LIN {X 0,Y 362.16,Z 503.994,A -85,B 0,C 180,E1 -13146.687,E2 -13146.687} C_VEL
LIN {X 0,Y 362.023,Z 504.013,A -85,B 0,C 180,E1 -13150.063,E2 -13150.063} C_VEL
LIN {X 0,Y 361.989,Z 504.018,A -85,B 0,C 180,E1 -13153.9,E2 -13153.9} C_VEL
LIN {X 0,Y 361.959,Z 504.022,A -85,B 0,C 180,E1 -13157.939,E2 -13157.939} C_VEL
LIN {X 0,Y 361.884,Z 504.034,A -85,B 0,C 180,E1 -13161.654,E2 -13161.654} C_VEL
LIN {X 0,Y 361.921,Z 504.028,A -85,B 0,C 180,E1 -13165.291,E2 -13165.291} C_VEL
LIN {X 0,Y 361.916,Z 504.029,A -85,B 0,C 180,E1 -13167.779,E2 -13167.779} C_VEL
LIN {X 0,Y 361.854,Z 504.038,A -85,B 0,C 180,E1 -13171.628,E2 -13171.628} C_VEL
LIN {X 0,Y 361.87,Z 504.035,A -85,B 0,C 180,E1 -13175.346,E2 -13175.346} C_VEL
LIN {X 0,Y 361.871,Z 504.032,A -85,B 0,C 180,E1 -13179.029,E2 -13179.029} C_VEL
LIN {X 0,Y 361.883,Z 504.029,A -85,B 0,C 180,E1 -13182.442,E2 -13182.442} C_VEL
LIN {X 0,Y 361.926,Z 504.026,A -85,B 0,C 180,E1 -13185.93,E2 -13185.93} C_VEL
LIN {X 0,Y 361.904,Z 504.029,A -85,B 0,C 180,E1 -13189.233,E2 -13189.233} C_VEL
LIN {X 0,Y 361.869,Z 504.032,A -85,B 0,C 180,E1 -13192.984,E2 -13192.984} C_VEL
LIN {X 0,Y 361.858,Z 504.032,A -85,B 0,C 180,E1 -13196.632,E2 -13196.632} C_VEL
LIN {X 0,Y 361.875,Z 504.036,A -85,B 0,C 180,E1 -13199.673,E2 -13199.673} C_VEL
LIN {X 0,Y 361.956,Z 504.025,A -85,B 0,C 180,E1 -13203.476,E2 -13203.476} C_VEL
LIN {X 0,Y 361.893,Z 504.03,A -85,B 0,C 180,E1 -13207.146,E2 -13207.146} C_VEL
LIN {X 0,Y 361.924,Z 504.024,A -85,B 0,C 180,E1 -13210.725,E2 -13210.725} C_VEL
LIN {X 0,Y 361.95,Z 504.021,A -85,B 0,C 180,E1 -13214.227,E2 -13214.227} C_VEL
LIN {X 0,Y 362.002,Z 504.014,A -85,B 0,C 180,E1 -13216.529,E2 -13216.529} C_VEL
LIN {X 0,Y 362.032,Z 504.013,A -85,B 0,C 180,E1 -13219.939,E2 -13219.939} C_VEL
LIN {X 0,Y 362.156,Z 503.998,A -85,B 0,C 180,E1 -13223.314,E2 -13223.314} C_VEL
LIN {X 0,Y 362.288,Z 503.983,A -85,B 0,C 180,E1 -13227.777,E2 -13227.777} C_VEL
LIN {X 0,Y 362.429,Z 503.963,A -85,B 0,C 180,E1 -13230.001,E2 -13230.001} C_VEL
LIN {X 0,Y 362.09,Z 504.004,A -85,B 0,C 180,E1 -13232.225,E2 -13232.225} C_VEL
LIN {X 0,Y 361.698,Z 504.058,A -85,B 0,C 180,E1 -13235.576,E2 -13235.576} C_VEL
LIN {X 0,Y 361.473,Z 504.131,A -85,B 0,C 180,E1 -13237.437,E2 -13237.437} C_VEL
LIN {X 0,Y 361.189,Z 507.102,A -85,B 0,C 180,E1 -13241.221,E2 -13241.221} C_VEL
LIN {X 0,Y 361.205,Z 507.651,A -85,B 0,C 180,E1 -13241.824,E2 -13241.824} C_VEL
LIN {X 0,Y 362.214,Z 510.606,A -85,B 0,C 180,E1 -13241.986,E2 -13241.986} C_VEL
LIN {X 0,Y 367.763,Z 525.518,A -85,B 0,C 180,E1 -13242.934,E2 -13242.934} C_VEL
LIN {X 0,Y 372.106,Z 539.202,A -85,B 0,C 180,E1 -13243.935,E2 -13243.935} C_VEL
LIN {X 0,Y 374.364,Z 547.439,A -85,B 0,C 180,E1 -13244.603,E2 -13244.603} C_VEL
LIN {X 0,Y 373.094,Z 561.384,A -85,B 0,C 180,E1 -13245.548,E2 -13245.548} C_VEL
LIN {X 0,Y 371.697,Z 574.147,A -85,B 0,C 180,E1 -13246.618,E2 -13246.618} C_VEL
LIN {X 0,Y 370.152,Z 586.321,A -85,B 0,C 180,E1 -13247.851,E2 -13247.851} C_VEL
LIN {X 0,Y 368.527,Z 598.526,A -85,B 0,C 180,E1 -13249.351,E2 -13249.351} C_VEL
LIN {X 0,Y 366.709,Z 610.314,A -85,B 0,C 180,E1 -13251.093,E2 -13251.093} C_VEL
LIN {X 0,Y 365.196,Z 620.6,A -85,B 0,C 180,E1 -13252.936,E2 -13252.936} C_VEL
LIN {X 0,Y 363.887,Z 629.278,A -85,B 0,C 180,E1 -13254.803,E2 -13254.803} C_VEL
LIN {X 0,Y 362.73,Z 637.566,A -85,B 0,C 180,E1 -13256.966,E2 -13256.966} C_VEL
LIN {X 0,Y 361.854,Z 644.084,A -85,B 0,C 180,E1 -13259.072,E2 -13259.072} C_VEL
LIN {X 0,Y 361.248,Z 649.166,A -85,B 0,C 180,E1 -13261.127,E2 -13261.127} C_VEL
LIN {X 0,Y 360.827,Z 653.239,A -85,B 0,C 180,E1 -13263.257,E2 -13263.257} C_VEL
LIN {X 0,Y 359.954,Z 654.717,A -85,B 0,C 180,E1 -13264.16,E2 -13264.16} C_VEL
LIN {X 0,Y 356.859,Z 656.726,A -85,B 0,C 180,E1 -13265.63,E2 -13265.63} C_VEL
LIN {X 0,Y 354.342,Z 657.99,A -85,B 0,C 180,E1 -13266.829,E2 -13266.829} C_VEL
LIN {X 0,Y 353.271,Z 658.718,A -85,B 0,C 180,E1 -13267.765,E2 -13267.765} C_VEL
LIN {X 0,Y 353.185,Z 658.865,A -85,B 0,C 180,E1 -13268.083,E2 -13268.083} C_VEL
LIN {X 0,Y 353.136,Z 659.368,A -85,B 0,C 180,E1 -13269.558,E2 -13269.558} C_VEL
LIN {X 0,Y 353.143,Z 659.407,A -85,B 0,C 180,E1 -13271.052,E2 -13271.052} C_VEL
LIN {X 0,Y 353.242,Z 658.953,A -85,B 0,C 180,E1 -13272.595,E2 -13272.595} C_VEL
LIN {X 0,Y 353.396,Z 657.843,A -85,B 0,C 180,E1 -13274.279,E2 -13274.279} C_VEL
LIN {X 0,Y 353.643,Z 656.133,A -85,B 0,C 180,E1 -13275.927,E2 -13275.927} C_VEL
LIN {X 0,Y 354.153,Z 652.64,A -85,B 0,C 180,E1 -13278.28,E2 -13278.28} C_VEL
LIN {X 0,Y 354.854,Z 647.717,A -85,B 0,C 180,E1 -13280.67,E2 -13280.67} C_VEL
LIN {X 0,Y 355.849,Z 641.498,A -85,B 0,C 180,E1 -13282.987,E2 -13282.987} C_VEL
LIN {X 0,Y 357.13,Z 634.019,A -85,B 0,C 180,E1 -13285.201,E2 -13285.201} C_VEL
LIN {X 0,Y 358.47,Z 626.29,A -85,B 0,C 180,E1 -13287.087,E2 -13287.087} C_VEL
LIN {X 0,Y 360.334,Z 616.189,A -85,B 0,C 180,E1 -13289.112,E2 -13289.112} C_VEL
LIN {X 0,Y 362.146,Z 605.801,A -85,B 0,C 180,E1 -13290.843,E2 -13290.843} C_VEL
LIN {X 0,Y 364.021,Z 594.626,A -85,B 0,C 180,E1 -13292.395,E2 -13292.395} C_VEL
LIN {X 0,Y 365.803,Z 582.756,A -85,B 0,C 180,E1 -13293.775,E2 -13293.775} C_VEL
LIN {X 0,Y 367.569,Z 569.94,A -85,B 0,C 180,E1 -13295.002,E2 -13295.002} C_VEL
LIN {X 0,Y 369.207,Z 556.741,A -85,B 0,C 180,E1 -13296.021,E2 -13296.021} C_VEL
LIN {X 0,Y 369.669,Z 552.277,A -85,B 0,C 180,E1 -13296.32,E2 -13296.32} C_VEL
LIN {X 0,Y 368.858,Z 548.08,A -85,B 0,C 180,E1 -13296.697,E2 -13296.697} C_VEL
LIN {X 0,Y 364.908,Z 535.544,A -85,B 0,C 180,E1 -13297.833,E2 -13297.833} C_VEL
LIN {X 0,Y 359.987,Z 523.202,A -85,B 0,C 180,E1 -13298.919,E2 -13298.919} C_VEL
LIN {X 0,Y 355.705,Z 514.122,A -85,B 0,C 180,E1 -13299.696,E2 -13299.696} C_VEL
LIN {X 0,Y 354.522,Z 510.981,A -85,B 0,C 180,E1 -13299.927,E2 -13299.927} C_VEL
LIN {X 0,Y 354.688,Z 509.194,A -85,B 0,C 180,E1 -13302.709,E2 -13302.709} C_VEL
LIN {X 0,Y 354.966,Z 507.016,A -85,B 0,C 180,E1 -13306.255,E2 -13306.255} C_VEL
LIN {X 0,Y 354.941,Z 505.058,A -85,B 0,C 180,E1 -13309.734,E2 -13309.734} C_VEL
LIN {X 0,Y 355.125,Z 504.875,A -85,B 0,C 180,E1 -13313.18,E2 -13313.18} C_VEL
LIN {X 0,Y 355.244,Z 504.861,A -85,B 0,C 180,E1 -13317.732,E2 -13317.732} C_VEL
LIN {X 0,Y 355.395,Z 504.84,A -85,B 0,C 180,E1 -13320,E2 -13320} C_VEL
LIN {X 0,Y 355.243,Z 504.86,A -85,B 0,C 180,E1 -13322.267,E2 -13322.267} C_VEL
LIN {X 0,Y 355.136,Z 504.873,A -85,B 0,C 180,E1 -13326.819,E2 -13326.819} C_VEL
LIN {X 0,Y 355.013,Z 504.887,A -85,B 0,C 180,E1 -13329.112,E2 -13329.112} C_VEL
LIN {X 0,Y 354.918,Z 504.902,A -85,B 0,C 180,E1 -13332.581,E2 -13332.581} C_VEL
LIN {X 0,Y 354.886,Z 504.903,A -85,B 0,C 180,E1 -13336.096,E2 -13336.096} C_VEL
LIN {X 0,Y 354.9,Z 504.905,A -85,B 0,C 180,E1 -13338.472,E2 -13338.472} C_VEL
LIN {X 0,Y 354.832,Z 504.911,A -85,B 0,C 180,E1 -13342.106,E2 -13342.106} C_VEL
LIN {X 0,Y 354.897,Z 504.904,A -85,B 0,C 180,E1 -13345.827,E2 -13345.827} C_VEL
LIN {X 0,Y 354.852,Z 504.91,A -85,B 0,C 180,E1 -13349.678,E2 -13349.678} C_VEL
LIN {X 0,Y 354.784,Z 504.919,A -85,B 0,C 180,E1 -13352.333,E2 -13352.333} C_VEL
LIN {X 0,Y 355.179,Z 506.831,A -85,B 0,C 180,E1 -13355.017,E2 -13355.017} C_VEL
LIN {X 0,Y 355.635,Z 509.455,A -85,B 0,C 180,E1 -13357.778,E2 -13357.778} C_VEL
LIN {X 0,Y 356.304,Z 513.425,A -85,B 0,C 180,E1 -13361.45,E2 -13361.45} C_VEL
LIN {X 0,Y 357.068,Z 517.953,A -85,B 0,C 180,E1 -13365.118,E2 -13365.118} C_VEL
LIN {X 0,Y 357.385,Z 520.082,A -85,B 0,C 180,E1 -13366.686,E2 -13366.686} C_VEL
LIN {X 0,Y 357.344,Z 522.48,A -85,B 0,C 180,E1 -13368.362,E2 -13368.362} C_VEL
LIN {X 0,Y 356.863,Z 526.472,A -85,B 0,C 180,E1 -13370.935,E2 -13370.935} C_VEL
LIN {X 0,Y 356.316,Z 531.446,A -85,B 0,C 180,E1 -13373.967,E2 -13373.967} C_VEL
LIN {X 0,Y 355.609,Z 538.026,A -85,B 0,C 180,E1 -13377.75,E2 -13377.75} C_VEL
LIN {X 0,Y 355.161,Z 542.305,A -85,B 0,C 180,E1 -13380.105,E2 -13380.105} C_VEL
LIN {X 0,Y 356.183,Z 545.901,A -85,B 0,C 180,E1 -13380.324,E2 -13380.324} C_VEL
LIN {X 0,Y 360.868,Z 561.008,A -85,B 0,C 180,E1 -13381.324,E2 -13381.324} C_VEL
LIN {X 0,Y 364.094,Z 575.482,A -85,B 0,C 180,E1 -13382.344,E2 -13382.344} C_VEL
LIN {X 0,Y 366.257,Z 589.592,A -85,B 0,C 180,E1 -13383.441,E2 -13383.441} C_VEL
LIN {X 0,Y 367.027,Z 598.105,A -85,B 0,C 180,E1 -13384.155,E2 -13384.155} C_VEL
LIN {X 0,Y 365.264,Z 611.753,A -85,B 0,C 180,E1 -13385.261,E2 -13385.261} C_VEL
LIN {X 0,Y 363.4,Z 624.255,A -85,B 0,C 180,E1 -13386.492,E2 -13386.492} C_VEL
LIN {X 0,Y 361.515,Z 635.974,A -85,B 0,C 180,E1 -13387.873,E2 -13387.873} C_VEL
LIN {X 0,Y 359.729,Z 646.937,A -85,B 0,C 180,E1 -13389.411,E2 -13389.411} C_VEL
LIN {X 0,Y 358.129,Z 657.131,A -85,B 0,C 180,E1 -13391.107,E2 -13391.107} C_VEL
LIN {X 0,Y 356.52,Z 667.138,A -85,B 0,C 180,E1 -13393.096,E2 -13393.096} C_VEL
LIN {X 0,Y 355.362,Z 675.529,A -85,B 0,C 180,E1 -13395.102,E2 -13395.102} C_VEL
LIN {X 0,Y 354.344,Z 683.421,A -85,B 0,C 180,E1 -13397.398,E2 -13397.398} C_VEL
LIN {X 0,Y 353.691,Z 689.735,A -85,B 0,C 180,E1 -13399.698,E2 -13399.698} C_VEL
LIN {X 0,Y 353.451,Z 694.63,A -85,B 0,C 180,E1 -13401.999,E2 -13401.999} C_VEL
LIN {X 0,Y 353.328,Z 698.216,A -85,B 0,C 180,E1 -13404.292,E2 -13404.292} C_VEL
LIN {X 0,Y 353.291,Z 700.57,A -85,B 0,C 180,E1 -13406.578,E2 -13406.578} C_VEL
LIN {X 0,Y 353.468,Z 701.749,A -85,B 0,C 180,E1 -13408.86,E2 -13408.86} C_VEL
LIN {X 0,Y 353.467,Z 701.745,A -85,B 0,C 180,E1 -13411.139,E2 -13411.139} C_VEL
LIN {X 0,Y 353.289,Z 700.5,A -85,B 0,C 180,E1 -13413.421,E2 -13413.421} C_VEL
LIN {X 0,Y 353.354,Z 698.05,A -85,B 0,C 180,E1 -13415.707,E2 -13415.707} C_VEL
LIN {X 0,Y 353.479,Z 694.348,A -85,B 0,C 180,E1 -13417.999,E2 -13417.999} C_VEL
LIN {X 0,Y 353.693,Z 689.298,A -85,B 0,C 180,E1 -13420.301,E2 -13420.301} C_VEL
LIN {X 0,Y 354.32,Z 682.788,A -85,B 0,C 180,E1 -13422.602,E2 -13422.602} C_VEL
LIN {X 0,Y 355.277,Z 674.631,A -85,B 0,C 180,E1 -13424.901,E2 -13424.901} C_VEL
LIN {X 0,Y 356.413,Z 665.932,A -85,B 0,C 180,E1 -13426.908,E2 -13426.908} C_VEL
LIN {X 0,Y 358.078,Z 655.484,A -85,B 0,C 180,E1 -13428.895,E2 -13428.895} C_VEL
LIN {X 0,Y 359.592,Z 644.775,A -85,B 0,C 180,E1 -13430.596,E2 -13430.596} C_VEL
LIN {X 0,Y 361.312,Z 633.147,A -85,B 0,C 180,E1 -13432.139,E2 -13432.139} C_VEL
LIN {X 0,Y 363.045,Z 620.511,A -85,B 0,C 180,E1 -13433.531,E2 -13433.531} C_VEL
LIN {X 0,Y 364.999,Z 606.726,A -85,B 0,C 180,E1 -13434.757,E2 -13434.757} C_VEL
LIN {X 0,Y 365.925,Z 597.042,A -85,B 0,C 180,E1 -13435.487,E2 -13435.487} C_VEL
LIN {X 0,Y 363.867,Z 582.779,A -85,B 0,C 180,E1 -13436.588,E2 -13436.588} C_VEL
LIN {X 0,Y 360.832,Z 567.462,A -85,B 0,C 180,E1 -13437.601,E2 -13437.601} C_VEL
LIN {X 0,Y 356.733,Z 551.393,A -85,B 0,C 180,E1 -13438.489,E2 -13438.489} C_VEL
LIN {X 0,Y 355.083,Z 545.125,A -85,B 0,C 180,E1 -13438.804,E2 -13438.804} C_VEL
LIN {X 0,Y 355.672,Z 538.75,A -85,B 0,C 180,E1 -13442.242,E2 -13442.242} C_VEL
LIN {X 0,Y 356.172,Z 533.916,A -85,B 0,C 180,E1 -13444.904,E2 -13444.904} C_VEL
LIN {X 0,Y 357.009,Z 526.725,A -85,B 0,C 180,E1 -13449.044,E2 -13449.044} C_VEL
LIN {X 0,Y 357.48,Z 521.886,A -85,B 0,C 180,E1 -13451.945,E2 -13451.945} C_VEL
LIN {X 0,Y 357.292,Z 518.352,A -85,B 0,C 180,E1 -13454.201,E2 -13454.201} C_VEL
LIN {X 0,Y 356.257,Z 513.007,A -85,B 0,C 180,E1 -13457.877,E2 -13457.877} C_VEL
LIN {X 0,Y 355.55,Z 509.052,A -85,B 0,C 180,E1 -13460.763,E2 -13460.763} C_VEL
LIN {X 0,Y 354.825,Z 504.91,A -85,B 0,C 180,E1 -13464.078,E2 -13464.078} C_VEL
LIN {X 0,Y 354.778,Z 504.918,A -85,B 0,C 180,E1 -13467.666,E2 -13467.666} C_VEL
LIN {X 0,Y 354.86,Z 504.903,A -85,B 0,C 180,E1 -13470.621,E2 -13470.621} C_VEL
LIN {X 0,Y 354.89,Z 504.901,A -85,B 0,C 180,E1 -13474.172,E2 -13474.172} C_VEL
LIN {X 0,Y 354.807,Z 504.913,A -85,B 0,C 180,E1 -13477.893,E2 -13477.893} C_VEL
LIN {X 0,Y 354.914,Z 504.899,A -85,B 0,C 180,E1 -13481.891,E2 -13481.891} C_VEL
LIN {X 0,Y 354.934,Z 504.896,A -85,B 0,C 180,E1 -13485.981,E2 -13485.981} C_VEL
LIN {X 0,Y 354.973,Z 504.893,A -85,B 0,C 180,E1 -13489.736,E2 -13489.736} C_VEL
LIN {X 0,Y 355.104,Z 504.874,A -85,B 0,C 180,E1 -13492.037,E2 -13492.037} C_VEL
LIN {X 0,Y 355.085,Z 504.876,A -85,B 0,C 180,E1 -13494.321,E2 -13494.321} C_VEL
LIN {X 0,Y 355.237,Z 504.861,A -85,B 0,C 180,E1 -13497.733,E2 -13497.733} C_VEL
LIN {X 0,Y 355.39,Z 504.839,A -85,B 0,C 180,E1 -13500,E2 -13500} C_VEL
LIN {X 0,Y 355.238,Z 504.857,A -85,B 0,C 180,E1 -13502.268,E2 -13502.268} C_VEL
LIN {X 0,Y 355.122,Z 504.871,A -85,B 0,C 180,E1 -13506.82,E2 -13506.82} C_VEL
LIN {X 0,Y 354.97,Z 504.89,A -85,B 0,C 180,E1 -13510.265,E2 -13510.265} C_VEL
LIN {X 0,Y 354.934,Z 504.896,A -85,B 0,C 180,E1 -13514.019,E2 -13514.019} C_VEL
LIN {X 0,Y 354.915,Z 504.898,A -85,B 0,C 180,E1 -13518.109,E2 -13518.109} C_VEL
LIN {X 0,Y 354.827,Z 504.909,A -85,B 0,C 180,E1 -13522.107,E2 -13522.107} C_VEL
LIN {X 0,Y 354.893,Z 504.903,A -85,B 0,C 180,E1 -13525.829,E2 -13525.829} C_VEL
LIN {X 0,Y 354.849,Z 504.91,A -85,B 0,C 180,E1 -13529.68,E2 -13529.68} C_VEL
LIN {X 0,Y 354.825,Z 504.913,A -85,B 0,C 180,E1 -13533.683,E2 -13533.683} C_VEL
LIN {X 0,Y 354.797,Z 504.911,A -85,B 0,C 180,E1 -13536.46,E2 -13536.46} C_VEL
LIN {X 0,Y 354.82,Z 504.913,A -85,B 0,C 180,E1 -13539.425,E2 -13539.425} C_VEL
LIN {X 0,Y 354.839,Z 504.907,A -85,B 0,C 180,E1 -13542.878,E2 -13542.878} C_VEL
LIN {X 0,Y 354.864,Z 504.904,A -85,B 0,C 180,E1 -13546.121,E2 -13546.121} C_VEL
LIN {X 0,Y 354.856,Z 504.906,A -85,B 0,C 180,E1 -13549.19,E2 -13549.19} C_VEL
LIN {X 0,Y 354.808,Z 504.91,A -85,B 0,C 180,E1 -13552.403,E2 -13552.403} C_VEL
LIN {X 0,Y 354.812,Z 504.91,A -85,B 0,C 180,E1 -13554.942,E2 -13554.942} C_VEL
LIN {X 0,Y 354.793,Z 504.912,A -85,B 0,C 180,E1 -13558.407,E2 -13558.407} C_VEL
LIN {X 0,Y 354.852,Z 504.911,A -85,B 0,C 180,E1 -13561.62,E2 -13561.62} C_VEL
LIN {X 0,Y 354.901,Z 504.899,A -85,B 0,C 180,E1 -13564.174,E2 -13564.174} C_VEL
LIN {X 0,Y 354.837,Z 504.91,A -85,B 0,C 180,E1 -13567.895,E2 -13567.895} C_VEL
LIN {X 0,Y 354.926,Z 504.899,A -85,B 0,C 180,E1 -13571.892,E2 -13571.892} C_VEL
LIN {X 0,Y 354.946,Z 504.895,A -85,B 0,C 180,E1 -13575.982,E2 -13575.982} C_VEL
LIN {X 0,Y 354.98,Z 504.894,A -85,B 0,C 180,E1 -13579.737,E2 -13579.737} C_VEL
LIN {X 0,Y 355.119,Z 504.873,A -85,B 0,C 180,E1 -13583.181,E2 -13583.181} C_VEL
LIN {X 0,Y 355.251,Z 504.86,A -85,B 0,C 180,E1 -13587.733,E2 -13587.733} C_VEL
LIN {X 0,Y 355.378,Z 504.842,A -85,B 0,C 180,E1 -13590.001,E2 -13590.001} C_VEL
LIN {X 0,Y 355.036,Z 504.882,A -85,B 0,C 180,E1 -13592.269,E2 -13592.269} C_VEL
LIN {X 0,Y 354.636,Z 504.938,A -85,B 0,C 180,E1 -13595.687,E2 -13595.687} C_VEL
LIN {X 0,Y 354.416,Z 505.032,A -85,B 0,C 180,E1 -13597.475,E2 -13597.475} C_VEL
LIN {X 0,Y 354.145,Z 508.008,A -85,B 0,C 180,E1 -13601.265,E2 -13601.265} C_VEL
LIN {X 0,Y 355.252,Z 511.174,A -85,B 0,C 180,E1 -13601.447,E2 -13601.447} C_VEL
LIN {X 0,Y 360.748,Z 525.852,A -85,B 0,C 180,E1 -13602.41,E2 -13602.41} C_VEL
LIN {X 0,Y 365.35,Z 540.123,A -85,B 0,C 180,E1 -13603.488,E2 -13603.488} C_VEL
LIN {X 0,Y 367.774,Z 549.128,A -85,B 0,C 180,E1 -13604.243,E2 -13604.243} C_VEL
LIN {X 0,Y 366.527,Z 562.147,A -85,B 0,C 180,E1 -13605.153,E2 -13605.153} C_VEL
LIN {X 0,Y 364.999,Z 575.512,A -85,B 0,C 180,E1 -13606.306,E2 -13606.306} C_VEL
LIN {X 0,Y 363.374,Z 587.771,A -85,B 0,C 180,E1 -13607.59,E2 -13607.59} C_VEL
LIN {X 0,Y 361.606,Z 600.088,A -85,B 0,C 180,E1 -13609.153,E2 -13609.153} C_VEL
LIN {X 0,Y 359.817,Z 611.407,A -85,B 0,C 180,E1 -13610.883,E2 -13610.883} C_VEL
LIN {X 0,Y 358.252,Z 621.651,A -85,B 0,C 180,E1 -13612.775,E2 -13612.775} C_VEL
LIN {X 0,Y 356.893,Z 630.347,A -85,B 0,C 180,E1 -13614.7,E2 -13614.7} C_VEL
LIN {X 0,Y 355.771,Z 637.841,A -85,B 0,C 180,E1 -13616.706,E2 -13616.706} C_VEL
LIN {X 0,Y 354.871,Z 644.367,A -85,B 0,C 180,E1 -13618.846,E2 -13618.846} C_VEL
LIN {X 0,Y 354.189,Z 649.739,A -85,B 0,C 180,E1 -13621.058,E2 -13621.058} C_VEL
LIN {X 0,Y 353.715,Z 654.107,A -85,B 0,C 180,E1 -13623.435,E2 -13623.435} C_VEL
LIN {X 0,Y 353.371,Z 656.7,A -85,B 0,C 180,E1 -13625.369,E2 -13625.369} C_VEL
LIN {X 0,Y 353.229,Z 658.374,A -85,B 0,C 180,E1 -13627.263,E2 -13627.263} C_VEL
LIN {X 0,Y 353.185,Z 658.865,A -85,B 0,C 180,E1 -13628.083,E2 -13628.083} C_VEL
LIN {X 0,Y 352.51,Z 659.364,A -85,B 0,C 180,E1 -13629.033,E2 -13629.033} C_VEL
LIN {X 0,Y 349.639,Z 659.804,A -85,B 0,C 180,E1 -13630.581,E2 -13630.581} C_VEL
LIN {X 0,Y 347.238,Z 659.718,A -85,B 0,C 180,E1 -13631.835,E2 -13631.835} C_VEL
LIN {X 0,Y 346.247,Z 659.345,A -85,B 0,C 180,E1 -13632.803,E2 -13632.803} C_VEL
LIN {X 0,Y 346.187,Z 659.154,A -85,B 0,C 180,E1 -13633.129,E2 -13633.129} C_VEL
LIN {X 0,Y 346.47,Z 657.522,A -85,B 0,C 180,E1 -13635.231,E2 -13635.231} C_VEL
LIN {X 0,Y 346.73,Z 655.615,A -85,B 0,C 180,E1 -13636.861,E2 -13636.861} C_VEL
LIN {X 0,Y 347.285,Z 652.028,A -85,B 0,C 180,E1 -13639.089,E2 -13639.089} C_VEL
LIN {X 0,Y 348.004,Z 647.43,A -85,B 0,C 180,E1 -13641.24,E2 -13641.24} C_VEL
LIN {X 0,Y 349.121,Z 640.92,A -85,B 0,C 180,E1 -13643.631,E2 -13643.631} C_VEL
LIN {X 0,Y 350.565,Z 633.311,A -85,B 0,C 180,E1 -13645.851,E2 -13645.851} C_VEL
LIN {X 0,Y 351.92,Z 625.632,A -85,B 0,C 180,E1 -13647.709,E2 -13647.709} C_VEL
LIN {X 0,Y 353.749,Z 616.337,A -85,B 0,C 180,E1 -13649.583,E2 -13649.583} C_VEL
LIN {X 0,Y 355.715,Z 605.713,A -85,B 0,C 180,E1 -13651.372,E2 -13651.372} C_VEL
LIN {X 0,Y 357.701,Z 594.358,A -85,B 0,C 180,E1 -13652.963,E2 -13652.963} C_VEL
LIN {X 0,Y 359.679,Z 581.843,A -85,B 0,C 180,E1 -13654.417,E2 -13654.417} C_VEL
LIN {X 0,Y 361.46,Z 569.204,A -85,B 0,C 180,E1 -13655.626,E2 -13655.626} C_VEL
LIN {X 0,Y 363.18,Z 555.577,A -85,B 0,C 180,E1 -13656.671,E2 -13656.671} C_VEL
LIN {X 0,Y 363.381,Z 553.731,A -85,B 0,C 180,E1 -13656.793,E2 -13656.793} C_VEL
LIN {X 0,Y 360.569,Z 543.123,A -85,B 0,C 180,E1 -13657.812,E2 -13657.812} C_VEL
LIN {X 0,Y 355.765,Z 529.842,A -85,B 0,C 180,E1 -13659.057,E2 -13659.057} C_VEL
LIN {X 0,Y 349.371,Z 515.614,A -85,B 0,C 180,E1 -13660.347,E2 -13660.347} C_VEL
LIN {X 0,Y 347.743,Z 512.591,A -85,B 0,C 180,E1 -13660.635,E2 -13660.635} C_VEL
LIN {X 0,Y 347.537,Z 511.513,A -85,B 0,C 180,E1 -13660.738,E2 -13660.738} C_VEL
LIN {X 0,Y 347.712,Z 509.757,A -85,B 0,C 180,E1 -13663.562,E2 -13663.562} C_VEL
LIN {X 0,Y 347.909,Z 508.314,A -85,B 0,C 180,E1 -13665.971,E2 -13665.971} C_VEL
LIN {X 0,Y 347.953,Z 506.342,A -85,B 0,C 180,E1 -13669.526,E2 -13669.526} C_VEL
LIN {X 0,Y 347.933,Z 505.773,A -85,B 0,C 180,E1 -13670.7,E2 -13670.7} C_VEL
LIN {X 0,Y 348.09,Z 505.751,A -85,B 0,C 180,E1 -13673.042,E2 -13673.042} C_VEL
LIN {X 0,Y 348.206,Z 505.738,A -85,B 0,C 180,E1 -13677.686,E2 -13677.686} C_VEL
LIN {X 0,Y 348.343,Z 505.719,A -85,B 0,C 180,E1 -13680,E2 -13680} C_VEL
LIN {X 0,Y 348.205,Z 505.737,A -85,B 0,C 180,E1 -13682.313,E2 -13682.313} C_VEL
LIN {X 0,Y 348.104,Z 505.748,A -85,B 0,C 180,E1 -13686.957,E2 -13686.957} C_VEL
LIN {X 0,Y 347.965,Z 505.764,A -85,B 0,C 180,E1 -13689.298,E2 -13689.298} C_VEL
LIN {X 0,Y 347.887,Z 505.775,A -85,B 0,C 180,E1 -13692.839,E2 -13692.839} C_VEL
LIN {X 0,Y 347.836,Z 505.784,A -85,B 0,C 180,E1 -13696.431,E2 -13696.431} C_VEL
LIN {X 0,Y 347.85,Z 505.779,A -85,B 0,C 180,E1 -13698.86,E2 -13698.86} C_VEL
LIN {X 0,Y 347.771,Z 505.79,A -85,B 0,C 180,E1 -13702.579,E2 -13702.579} C_VEL
LIN {X 0,Y 347.809,Z 505.783,A -85,B 0,C 180,E1 -13705.108,E2 -13705.108} C_VEL
LIN {X 0,Y 347.81,Z 505.788,A -85,B 0,C 180,E1 -13707.694,E2 -13707.694} C_VEL
LIN {X 0,Y 347.762,Z 505.792,A -85,B 0,C 180,E1 -13710.346,E2 -13710.346} C_VEL
LIN {X 0,Y 347.753,Z 505.922,A -85,B 0,C 180,E1 -13711.918,E2 -13711.918} C_VEL
LIN {X 0,Y 348.39,Z 509.086,A -85,B 0,C 180,E1 -13715.803,E2 -13715.803} C_VEL
LIN {X 0,Y 348.841,Z 511.83,A -85,B 0,C 180,E1 -13718.649,E2 -13718.649} C_VEL
LIN {X 0,Y 349.446,Z 515.405,A -85,B 0,C 180,E1 -13721.915,E2 -13721.915} C_VEL
LIN {X 0,Y 350.153,Z 519.638,A -85,B 0,C 180,E1 -13725.373,E2 -13725.373} C_VEL
LIN {X 0,Y 350.386,Z 523.089,A -85,B 0,C 180,E1 -13727.914,E2 -13727.914} C_VEL
LIN {X 0,Y 349.882,Z 527.362,A -85,B 0,C 180,E1 -13730.748,E2 -13730.748} C_VEL
LIN {X 0,Y 349.211,Z 533.058,A -85,B 0,C 180,E1 -13734.293,E2 -13734.293} C_VEL
LIN {X 0,Y 348.542,Z 539.153,A -85,B 0,C 180,E1 -13737.874,E2 -13737.874} C_VEL
LIN {X 0,Y 348.231,Z 541.767,A -85,B 0,C 180,E1 -13739.353,E2 -13739.353} C_VEL
LIN {X 0,Y 349.212,Z 545.248,A -85,B 0,C 180,E1 -13739.574,E2 -13739.574} C_VEL
LIN {X 0,Y 354.033,Z 560.283,A -85,B 0,C 180,E1 -13740.624,E2 -13740.624} C_VEL
LIN {X 0,Y 357.251,Z 574.069,A -85,B 0,C 180,E1 -13741.647,E2 -13741.647} C_VEL
LIN {X 0,Y 359.358,Z 587.189,A -85,B 0,C 180,E1 -13742.692,E2 -13742.692} C_VEL
LIN {X 0,Y 360.517,Z 599.249,A -85,B 0,C 180,E1 -13743.732,E2 -13743.732} C_VEL
LIN {X 0,Y 358.582,Z 613.339,A -85,B 0,C 180,E1 -13744.923,E2 -13744.923} C_VEL
LIN {X 0,Y 356.468,Z 626.728,A -85,B 0,C 180,E1 -13746.315,E2 -13746.315} C_VEL
LIN {X 0,Y 354.363,Z 639.018,A -85,B 0,C 180,E1 -13747.863,E2 -13747.863} C_VEL
LIN {X 0,Y 352.359,Z 650.631,A -85,B 0,C 180,E1 -13749.625,E2 -13749.625} C_VEL
LIN {X 0,Y 350.608,Z 661.387,A -85,B 0,C 180,E1 -13751.596,E2 -13751.596} C_VEL
LIN {X 0,Y 349.071,Z 670.628,A -85,B 0,C 180,E1 -13753.628,E2 -13753.628} C_VEL
LIN {X 0,Y 347.764,Z 679.351,A -85,B 0,C 180,E1 -13755.965,E2 -13755.965} C_VEL
LIN {X 0,Y 346.985,Z 686.404,A -85,B 0,C 180,E1 -13758.314,E2 -13758.314} C_VEL
LIN {X 0,Y 346.496,Z 691.976,A -85,B 0,C 180,E1 -13760.661,E2 -13760.661} C_VEL
LIN {X 0,Y 346.304,Z 696.192,A -85,B 0,C 180,E1 -13763.006,E2 -13763.006} C_VEL
LIN {X 0,Y 346.241,Z 699.141,A -85,B 0,C 180,E1 -13765.342,E2 -13765.342} C_VEL
LIN {X 0,Y 346.292,Z 700.887,A -85,B 0,C 180,E1 -13767.673,E2 -13767.673} C_VEL
LIN {X 0,Y 346.397,Z 701.46,A -85,B 0,C 180,E1 -13769.999,E2 -13769.999} C_VEL
LIN {X 0,Y 346.403,Z 701.304,A -85,B 0,C 180,E1 -13771.162,E2 -13771.162} C_VEL
LIN {X 0,Y 346.211,Z 700.05,A -85,B 0,C 180,E1 -13773.491,E2 -13773.491} C_VEL
LIN {X 0,Y 346.322,Z 697.252,A -85,B 0,C 180,E1 -13776.086,E2 -13776.086} C_VEL
LIN {X 0,Y 346.391,Z 693.852,A -85,B 0,C 180,E1 -13778.164,E2 -13778.164} C_VEL
LIN {X 0,Y 346.641,Z 688.778,A -85,B 0,C 180,E1 -13780.513,E2 -13780.513} C_VEL
LIN {X 0,Y 347.304,Z 682.24,A -85,B 0,C 180,E1 -13782.861,E2 -13782.861} C_VEL
LIN {X 0,Y 348.334,Z 674.055,A -85,B 0,C 180,E1 -13785.205,E2 -13785.205} C_VEL
LIN {X 0,Y 349.534,Z 665.322,A -85,B 0,C 180,E1 -13787.251,E2 -13787.251} C_VEL
LIN {X 0,Y 351.226,Z 654.831,A -85,B 0,C 180,E1 -13789.278,E2 -13789.278} C_VEL
LIN {X 0,Y 352.837,Z 644.079,A -85,B 0,C 180,E1 -13791.009,E2 -13791.009} C_VEL
LIN {X 0,Y 354.666,Z 632.4,A -85,B 0,C 180,E1 -13792.576,E2 -13792.576} C_VEL
LIN {X 0,Y 356.496,Z 619.7,A -85,B 0,C 180,E1 -13793.991,E2 -13793.991} C_VEL
LIN {X 0,Y 358.491,Z 605.825,A -85,B 0,C 180,E1 -13795.238,E2 -13795.238} C_VEL
LIN {X 0,Y 359.217,Z 598.016,A -85,B 0,C 180,E1 -13795.845,E2 -13795.845} C_VEL
LIN {X 0,Y 357.268,Z 584.061,A -85,B 0,C 180,E1 -13796.968,E2 -13796.968} C_VEL
LIN {X 0,Y 354.357,Z 569.115,A -85,B 0,C 180,E1 -13798.002,E2 -13798.002} C_VEL
LIN {X 0,Y 350.526,Z 553.68,A -85,B 0,C 180,E1 -13798.91,E2 -13798.91} C_VEL
LIN {X 0,Y 348.097,Z 544.696,A -85,B 0,C 180,E1 -13799.387,E2 -13799.387} C_VEL
LIN {X 0,Y 348.769,Z 538.235,A -85,B 0,C 180,E1 -13802.96,E2 -13802.96} C_VEL
LIN {X 0,Y 349.359,Z 532.232,A -85,B 0,C 180,E1 -13806.422,E2 -13806.422} C_VEL
LIN {X 0,Y 350.157,Z 526.238,A -85,B 0,C 180,E1 -13809.96,E2 -13809.96} C_VEL
LIN {X 0,Y 350.482,Z 522.766,A -85,B 0,C 180,E1 -13812.104,E2 -13812.104} C_VEL
LIN {X 0,Y 350.198,Z 518.941,A -85,B 0,C 180,E1 -13814.618,E2 -13814.618} C_VEL
LIN {X 0,Y 349.181,Z 513.608,A -85,B 0,C 180,E1 -13818.38,E2 -13818.38} C_VEL
LIN {X 0,Y 348.141,Z 507.896,A -85,B 0,C 180,E1 -13822.727,E2 -13822.727} C_VEL
LIN {X 0,Y 347.787,Z 505.787,A -85,B 0,C 180,E1 -13824.481,E2 -13824.481} C_VEL
LIN {X 0,Y 347.736,Z 505.791,A -85,B 0,C 180,E1 -13828.3,E2 -13828.3} C_VEL
LIN {X 0,Y 347.797,Z 505.785,A -85,B 0,C 180,E1 -13830.99,E2 -13830.99} C_VEL
LIN {X 0,Y 347.823,Z 505.786,A -85,B 0,C 180,E1 -13833.607,E2 -13833.607} C_VEL
LIN {X 0,Y 347.776,Z 505.787,A -85,B 0,C 180,E1 -13836.161,E2 -13836.161} C_VEL
LIN {X 0,Y 347.802,Z 505.785,A -85,B 0,C 180,E1 -13839.909,E2 -13839.909} C_VEL
LIN {X 0,Y 347.858,Z 505.776,A -85,B 0,C 180,E1 -13842.359,E2 -13842.359} C_VEL
LIN {X 0,Y 347.888,Z 505.774,A -85,B 0,C 180,E1 -13845.971,E2 -13845.971} C_VEL
LIN {X 0,Y 347.923,Z 505.773,A -85,B 0,C 180,E1 -13849.526,E2 -13849.526} C_VEL
LIN {X 0,Y 348.064,Z 505.752,A -85,B 0,C 180,E1 -13851.875,E2 -13851.875} C_VEL
LIN {X 0,Y 348.06,Z 505.751,A -85,B 0,C 180,E1 -13854.206,E2 -13854.206} C_VEL
LIN {X 0,Y 348.2,Z 505.737,A -85,B 0,C 180,E1 -13857.687,E2 -13857.687} C_VEL
LIN {X 0,Y 348.338,Z 505.716,A -85,B 0,C 180,E1 -13860,E2 -13860} C_VEL
LIN {X 0,Y 348.201,Z 505.732,A -85,B 0,C 180,E1 -13862.314,E2 -13862.314} C_VEL
LIN {X 0,Y 348.087,Z 505.748,A -85,B 0,C 180,E1 -13866.959,E2 -13866.959} C_VEL
LIN {X 0,Y 347.92,Z 505.767,A -85,B 0,C 180,E1 -13870.475,E2 -13870.475} C_VEL
LIN {X 0,Y 347.89,Z 505.772,A -85,B 0,C 180,E1 -13874.151,E2 -13874.151} C_VEL
LIN {X 0,Y 347.883,Z 505.773,A -85,B 0,C 180,E1 -13878.291,E2 -13878.291} C_VEL
LIN {X 0,Y 347.781,Z 505.79,A -85,B 0,C 180,E1 -13881.636,E2 -13881.636} C_VEL
LIN {X 0,Y 347.805,Z 505.783,A -85,B 0,C 180,E1 -13885.11,E2 -13885.11} C_VEL
LIN {X 0,Y 347.806,Z 505.787,A -85,B 0,C 180,E1 -13887.695,E2 -13887.695} C_VEL
LIN {X 0,Y 347.765,Z 505.788,A -85,B 0,C 180,E1 -13890.347,E2 -13890.347} C_VEL
LIN {X 0,Y 347.743,Z 505.791,A -85,B 0,C 180,E1 -13894.045,E2 -13894.045} C_VEL
LIN {X 0,Y 347.762,Z 505.79,A -85,B 0,C 180,E1 -13897.321,E2 -13897.321} C_VEL
LIN {X 0,Y 347.79,Z 505.785,A -85,B 0,C 180,E1 -13900.29,E2 -13900.29} C_VEL
LIN {X 0,Y 347.816,Z 505.785,A -85,B 0,C 180,E1 -13903.394,E2 -13903.394} C_VEL
LIN {X 0,Y 347.815,Z 505.78,A -85,B 0,C 180,E1 -13906.671,E2 -13906.671} C_VEL
LIN {X 0,Y 347.784,Z 505.786,A -85,B 0,C 180,E1 -13910.167,E2 -13910.167} C_VEL
LIN {X 0,Y 347.789,Z 505.785,A -85,B 0,C 180,E1 -13914.126,E2 -13914.126} C_VEL
LIN {X 0,Y 347.738,Z 505.793,A -85,B 0,C 180,E1 -13918.087,E2 -13918.087} C_VEL
LIN {X 0,Y 347.806,Z 505.783,A -85,B 0,C 180,E1 -13920.991,E2 -13920.991} C_VEL
LIN {X 0,Y 347.834,Z 505.784,A -85,B 0,C 180,E1 -13923.609,E2 -13923.609} C_VEL
LIN {X 0,Y 347.79,Z 505.786,A -85,B 0,C 180,E1 -13926.163,E2 -13926.163} C_VEL
LIN {X 0,Y 347.82,Z 505.783,A -85,B 0,C 180,E1 -13929.911,E2 -13929.911} C_VEL
LIN {X 0,Y 347.87,Z 505.775,A -85,B 0,C 180,E1 -13932.36,E2 -13932.36} C_VEL
LIN {X 0,Y 347.901,Z 505.773,A -85,B 0,C 180,E1 -13935.972,E2 -13935.972} C_VEL
LIN {X 0,Y 347.931,Z 505.772,A -85,B 0,C 180,E1 -13939.526,E2 -13939.526} C_VEL
LIN {X 0,Y 348.084,Z 505.749,A -85,B 0,C 180,E1 -13943.043,E2 -13943.043} C_VEL
LIN {X 0,Y 348.214,Z 505.737,A -85,B 0,C 180,E1 -13947.687,E2 -13947.687} C_VEL
LIN {X 0,Y 348.327,Z 505.72,A -85,B 0,C 180,E1 -13950.001,E2 -13950.001} C_VEL
LIN {X 0,Y 347.984,Z 505.761,A -85,B 0,C 180,E1 -13952.316,E2 -13952.316} C_VEL
LIN {X 0,Y 347.577,Z 505.816,A -85,B 0,C 180,E1 -13955.803,E2 -13955.803} C_VEL
LIN {X 0,Y 347.377,Z 505.961,A -85,B 0,C 180,E1 -13957.536,E2 -13957.536} C_VEL
LIN {X 0,Y 347.121,Z 508.375,A -85,B 0,C 180,E1 -13960.684,E2 -13960.684} C_VEL
LIN {X 0,Y 348.204,Z 511.585,A -85,B 0,C 180,E1 -13960.871,E2 -13960.871} C_VEL
LIN {X 0,Y 353.743,Z 525.985,A -85,B 0,C 180,E1 -13961.859,E2 -13961.859} C_VEL
LIN {X 0,Y 358.204,Z 539.631,A -85,B 0,C 180,E1 -13962.914,E2 -13962.914} C_VEL
LIN {X 0,Y 361.075,Z 550.27,A -85,B 0,C 180,E1 -13963.826,E2 -13963.826} C_VEL
LIN {X 0,Y 360.827,Z 555.319,A -85,B 0,C 180,E1 -13964.182,E2 -13964.182} C_VEL
LIN {X 0,Y 359.143,Z 569.797,A -85,B 0,C 180,E1 -13965.318,E2 -13965.318} C_VEL
LIN {X 0,Y 357.356,Z 583.557,A -85,B 0,C 180,E1 -13966.672,E2 -13966.672} C_VEL
LIN {X 0,Y 355.566,Z 596.378,A -85,B 0,C 180,E1 -13968.224,E2 -13968.224} C_VEL
LIN {X 0,Y 353.817,Z 606.881,A -85,B 0,C 180,E1 -13969.736,E2 -13969.736} C_VEL
LIN {X 0,Y 352.306,Z 616.366,A -85,B 0,C 180,E1 -13971.35,E2 -13971.35} C_VEL
LIN {X 0,Y 350.82,Z 625.639,A -85,B 0,C 180,E1 -13973.232,E2 -13973.232} C_VEL
LIN {X 0,Y 349.497,Z 633.681,A -85,B 0,C 180,E1 -13975.188,E2 -13975.188} C_VEL
LIN {X 0,Y 348.287,Z 641.961,A -85,B 0,C 180,E1 -13977.653,E2 -13977.653} C_VEL
LIN {X 0,Y 347.548,Z 647.167,A -85,B 0,C 180,E1 -13979.594,E2 -13979.594} C_VEL
LIN {X 0,Y 346.982,Z 651.873,A -85,B 0,C 180,E1 -13981.777,E2 -13981.777} C_VEL
LIN {X 0,Y 346.566,Z 655.175,A -85,B 0,C 180,E1 -13983.752,E2 -13983.752} C_VEL
LIN {X 0,Y 346.202,Z 657.872,A -85,B 0,C 180,E1 -13986.065,E2 -13986.065} C_VEL
LIN {X 0,Y 346.084,Z 659.276,A -85,B 0,C 180,E1 -13988.069,E2 -13988.069} C_VEL
LIN {X 0,Y 346.065,Z 659.782,A -85,B 0,C 180,E1 -13989.491,E2 -13989.491} C_VEL
LIN {X 0,Y 346.095,Z 659.611,A -85,B 0,C 180,E1 -13992.076,E2 -13992.076} C_VEL
LIN {X 0,Y 346.187,Z 659.154,A -85,B 0,C 180,E1 -13993.129,E2 -13993.129} C_VEL
LIN {X 0,Y 345.622,Z 658.586,A -85,B 0,C 180,E1 -13994.098,E2 -13994.098} C_VEL
LIN {X 0,Y 343.009,Z 657.38,A -85,B 0,C 180,E1 -13995.679,E2 -13995.679} C_VEL
LIN {X 0,Y 340.842,Z 656.114,A -85,B 0,C 180,E1 -13996.948,E2 -13996.948} C_VEL
LIN {X 0,Y 340.013,Z 654.824,A -85,B 0,C 180,E1 -13997.913,E2 -13997.913} C_VEL
LIN {X 0,Y 340,Z 654.314,A -85,B 0,C 180,E1 -13998.236,E2 -13998.236} C_VEL
LIN {X 0,Y 340.837,Z 649.211,A -85,B 0,C 180,E1 -14000.937,E2 -14000.937} C_VEL
LIN {X 0,Y 341.959,Z 642.958,A -85,B 0,C 180,E1 -14003.414,E2 -14003.414} C_VEL
LIN {X 0,Y 343.453,Z 635.329,A -85,B 0,C 180,E1 -14005.792,E2 -14005.792} C_VEL
LIN {X 0,Y 345.17,Z 626.434,A -85,B 0,C 180,E1 -14008.035,E2 -14008.035} C_VEL
LIN {X 0,Y 347.159,Z 616.727,A -85,B 0,C 180,E1 -14010.036,E2 -14010.036} C_VEL
LIN {X 0,Y 349.205,Z 606.199,A -85,B 0,C 180,E1 -14011.838,E2 -14011.838} C_VEL
LIN {X 0,Y 351.213,Z 595.281,A -85,B 0,C 180,E1 -14013.401,E2 -14013.401} C_VEL
LIN {X 0,Y 353.216,Z 583.299,A -85,B 0,C 180,E1 -14014.83,E2 -14014.83} C_VEL
LIN {X 0,Y 355.141,Z 570.303,A -85,B 0,C 180,E1 -14016.108,E2 -14016.108} C_VEL
LIN {X 0,Y 357.027,Z 556.087,A -85,B 0,C 180,E1 -14017.226,E2 -14017.226} C_VEL
LIN {X 0,Y 356.711,Z 553.599,A -85,B 0,C 180,E1 -14017.452,E2 -14017.452} C_VEL
LIN {X 0,Y 352.668,Z 540.027,A -85,B 0,C 180,E1 -14018.821,E2 -14018.821} C_VEL
LIN {X 0,Y 347.331,Z 526.503,A -85,B 0,C 180,E1 -14020.15,E2 -14020.15} C_VEL
LIN {X 0,Y 341.864,Z 515.429,A -85,B 0,C 180,E1 -14021.231,E2 -14021.231} C_VEL
LIN {X 0,Y 340.74,Z 512.942,A -85,B 0,C 180,E1 -14021.453,E2 -14021.453} C_VEL
LIN {X 0,Y 340.589,Z 512.073,A -85,B 0,C 180,E1 -14021.548,E2 -14021.548} C_VEL
LIN {X 0,Y 340.869,Z 509.612,A -85,B 0,C 180,E1 -14025.704,E2 -14025.704} C_VEL
LIN {X 0,Y 340.936,Z 507.647,A -85,B 0,C 180,E1 -14029.308,E2 -14029.308} C_VEL
LIN {X 0,Y 340.998,Z 506.636,A -85,B 0,C 180,E1 -14031.704,E2 -14031.704} C_VEL
LIN {X 0,Y 341.038,Z 506.63,A -85,B 0,C 180,E1 -14034.085,E2 -14034.085} C_VEL
LIN {X 0,Y 341.168,Z 506.615,A -85,B 0,C 180,E1 -14037.638,E2 -14037.638} C_VEL
LIN {X 0,Y 341.294,Z 506.597,A -85,B 0,C 180,E1 -14040,E2 -14040} C_VEL
LIN {X 0,Y 341.167,Z 506.614,A -85,B 0,C 180,E1 -14042.361,E2 -14042.361} C_VEL
LIN {X 0,Y 341.073,Z 506.623,A -85,B 0,C 180,E1 -14047.101,E2 -14047.101} C_VEL
LIN {X 0,Y 340.868,Z 506.65,A -85,B 0,C 180,E1 -14050.693,E2 -14050.693} C_VEL
LIN {X 0,Y 340.861,Z 506.651,A -85,B 0,C 180,E1 -14054.325,E2 -14054.325} C_VEL
LIN {X 0,Y 340.835,Z 506.657,A -85,B 0,C 180,E1 -14058.466,E2 -14058.466} C_VEL
LIN {X 0,Y 340.751,Z 506.664,A -85,B 0,C 180,E1 -14061.857,E2 -14061.857} C_VEL
LIN {X 0,Y 340.77,Z 506.663,A -85,B 0,C 180,E1 -14065.664,E2 -14065.664} C_VEL
LIN {X 0,Y 340.74,Z 506.666,A -85,B 0,C 180,E1 -14068.319,E2 -14068.319} C_VEL
LIN {X 0,Y 340.741,Z 506.888,A -85,B 0,C 180,E1 -14071.04,E2 -14071.04} C_VEL
LIN {X 0,Y 341.335,Z 510.104,A -85,B 0,C 180,E1 -14075.205,E2 -14075.205} C_VEL
LIN {X 0,Y 341.922,Z 513.307,A -85,B 0,C 180,E1 -14078.642,E2 -14078.642} C_VEL
LIN {X 0,Y 342.564,Z 517.375,A -85,B 0,C 180,E1 -14082.39,E2 -14082.39} C_VEL
LIN {X 0,Y 343.28,Z 521.618,A -85,B 0,C 180,E1 -14085.886,E2 -14085.886} C_VEL
LIN {X 0,Y 343.346,Z 524.891,A -85,B 0,C 180,E1 -14088.299,E2 -14088.299} C_VEL
LIN {X 0,Y 342.62,Z 530.476,A -85,B 0,C 180,E1 -14092.021,E2 -14092.021} C_VEL
LIN {X 0,Y 341.972,Z 535.718,A -85,B 0,C 180,E1 -14095.29,E2 -14095.29} C_VEL
LIN {X 0,Y 341.35,Z 541.369,A -85,B 0,C 180,E1 -14098.567,E2 -14098.567} C_VEL
LIN {X 0,Y 342.369,Z 544.839,A -85,B 0,C 180,E1 -14098.791,E2 -14098.791} C_VEL
LIN {X 0,Y 347.259,Z 559.731,A -85,B 0,C 180,E1 -14099.904,E2 -14099.904} C_VEL
LIN {X 0,Y 350.374,Z 572.655,A -85,B 0,C 180,E1 -14100.904,E2 -14100.904} C_VEL
LIN {X 0,Y 352.787,Z 587.034,A -85,B 0,C 180,E1 -14102.094,E2 -14102.094} C_VEL
LIN {X 0,Y 354.013,Z 600.334,A -85,B 0,C 180,E1 -14103.298,E2 -14103.298} C_VEL
LIN {X 0,Y 352.156,Z 613.36,A -85,B 0,C 180,E1 -14104.433,E2 -14104.433} C_VEL
LIN {X 0,Y 349.958,Z 626.664,A -85,B 0,C 180,E1 -14105.847,E2 -14105.847} C_VEL
LIN {X 0,Y 347.766,Z 638.891,A -85,B 0,C 180,E1 -14107.42,E2 -14107.42} C_VEL
LIN {X 0,Y 345.741,Z 649.957,A -85,B 0,C 180,E1 -14109.13,E2 -14109.13} C_VEL
LIN {X 0,Y 343.813,Z 661.121,A -85,B 0,C 180,E1 -14111.219,E2 -14111.219} C_VEL
LIN {X 0,Y 342.198,Z 670.332,A -85,B 0,C 180,E1 -14113.29,E2 -14113.29} C_VEL
LIN {X 0,Y 340.804,Z 679.023,A -85,B 0,C 180,E1 -14115.672,E2 -14115.672} C_VEL
LIN {X 0,Y 339.969,Z 686.057,A -85,B 0,C 180,E1 -14118.069,E2 -14118.069} C_VEL
LIN {X 0,Y 339.415,Z 691.612,A -85,B 0,C 180,E1 -14120.465,E2 -14120.465} C_VEL
LIN {X 0,Y 339.226,Z 695.806,A -85,B 0,C 180,E1 -14122.859,E2 -14122.859} C_VEL
LIN {X 0,Y 339.156,Z 698.738,A -85,B 0,C 180,E1 -14125.245,E2 -14125.245} C_VEL
LIN {X 0,Y 339.195,Z 700.469,A -85,B 0,C 180,E1 -14127.624,E2 -14127.624} C_VEL
LIN {X 0,Y 339.336,Z 701.028,A -85,B 0,C 180,E1 -14129.999,E2 -14129.999} C_VEL
LIN {X 0,Y 339.197,Z 700.389,A -85,B 0,C 180,E1 -14132.374,E2 -14132.374} C_VEL
LIN {X 0,Y 339.185,Z 698.509,A -85,B 0,C 180,E1 -14134.753,E2 -14134.753} C_VEL
LIN {X 0,Y 339.241,Z 695.395,A -85,B 0,C 180,E1 -14137.14,E2 -14137.14} C_VEL
LIN {X 0,Y 339.417,Z 690.984,A -85,B 0,C 180,E1 -14139.534,E2 -14139.534} C_VEL
LIN {X 0,Y 339.954,Z 685.174,A -85,B 0,C 180,E1 -14141.93,E2 -14141.93} C_VEL
LIN {X 0,Y 340.766,Z 677.804,A -85,B 0,C 180,E1 -14144.328,E2 -14144.328} C_VEL
LIN {X 0,Y 341.9,Z 669.92,A -85,B 0,C 180,E1 -14146.417,E2 -14146.417} C_VEL
LIN {X 0,Y 343.437,Z 660.45,A -85,B 0,C 180,E1 -14148.492,E2 -14148.492} C_VEL
LIN {X 0,Y 344.994,Z 650.814,A -85,B 0,C 180,E1 -14150.261,E2 -14150.261} C_VEL
LIN {X 0,Y 346.798,Z 639.374,A -85,B 0,C 180,E1 -14152.018,E2 -14152.018} C_VEL
LIN {X 0,Y 348.832,Z 626.841,A -85,B 0,C 180,E1 -14153.604,E2 -14153.604} C_VEL
LIN {X 0,Y 350.389,Z 615.996,A -85,B 0,C 180,E1 -14154.752,E2 -14154.752} C_VEL
LIN {X 0,Y 352.211,Z 603.229,A -85,B 0,C 180,E1 -14155.868,E2 -14155.868} C_VEL
LIN {X 0,Y 352.511,Z 598.964,A -85,B 0,C 180,E1 -14156.213,E2 -14156.213} C_VEL
LIN {X 0,Y 350.403,Z 583.802,A -85,B 0,C 180,E1 -14157.47,E2 -14157.47} C_VEL
LIN {X 0,Y 347.365,Z 568.285,A -85,B 0,C 180,E1 -14158.573,E2 -14158.573} C_VEL
LIN {X 0,Y 343.391,Z 552.653,A -85,B 0,C 180,E1 -14159.523,E2 -14159.523} C_VEL
LIN {X 0,Y 341.136,Z 544.307,A -85,B 0,C 180,E1 -14159.984,E2 -14159.984} C_VEL
LIN {X 0,Y 341.848,Z 537.775,A -85,B 0,C 180,E1 -14163.715,E2 -14163.715} C_VEL
LIN {X 0,Y 342.382,Z 532.476,A -85,B 0,C 180,E1 -14166.818,E2 -14166.818} C_VEL
LIN {X 0,Y 343.143,Z 527.1,A -85,B 0,C 180,E1 -14170.085,E2 -14170.085} C_VEL
LIN {X 0,Y 343.449,Z 523.192,A -85,B 0,C 180,E1 -14172.552,E2 -14172.552} C_VEL
LIN {X 0,Y 343.082,Z 519.525,A -85,B 0,C 180,E1 -14175.031,E2 -14175.031} C_VEL
LIN {X 0,Y 342.043,Z 514.222,A -85,B 0,C 180,E1 -14178.89,E2 -14178.89} C_VEL
LIN {X 0,Y 341.369,Z 510.369,A -85,B 0,C 180,E1 -14181.857,E2 -14181.857} C_VEL
LIN {X 0,Y 340.71,Z 506.669,A -85,B 0,C 180,E1 -14184.968,E2 -14184.968} C_VEL
LIN {X 0,Y 340.695,Z 506.67,A -85,B 0,C 180,E1 -14188.956,E2 -14188.956} C_VEL
LIN {X 0,Y 340.771,Z 506.659,A -85,B 0,C 180,E1 -14192.473,E2 -14192.473} C_VEL
LIN {X 0,Y 340.745,Z 506.667,A -85,B 0,C 180,E1 -14195.638,E2 -14195.638} C_VEL
LIN {X 0,Y 340.728,Z 506.67,A -85,B 0,C 180,E1 -14199.473,E2 -14199.473} C_VEL
LIN {X 0,Y 340.849,Z 506.651,A -85,B 0,C 180,E1 -14201.984,E2 -14201.984} C_VEL
LIN {X 0,Y 340.86,Z 506.652,A -85,B 0,C 180,E1 -14205.705,E2 -14205.705} C_VEL
LIN {X 0,Y 340.866,Z 506.65,A -85,B 0,C 180,E1 -14209.306,E2 -14209.306} C_VEL
LIN {X 0,Y 341.066,Z 506.622,A -85,B 0,C 180,E1 -14212.898,E2 -14212.898} C_VEL
LIN {X 0,Y 341.162,Z 506.614,A -85,B 0,C 180,E1 -14217.639,E2 -14217.639} C_VEL
LIN {X 0,Y 341.289,Z 506.593,A -85,B 0,C 180,E1 -14220,E2 -14220} C_VEL
LIN {X 0,Y 341.163,Z 506.608,A -85,B 0,C 180,E1 -14222.362,E2 -14222.362} C_VEL
LIN {X 0,Y 341.054,Z 506.625,A -85,B 0,C 180,E1 -14227.103,E2 -14227.103} C_VEL
LIN {X 0,Y 340.863,Z 506.645,A -85,B 0,C 180,E1 -14230.695,E2 -14230.695} C_VEL
LIN {X 0,Y 340.855,Z 506.647,A -85,B 0,C 180,E1 -14234.326,E2 -14234.326} C_VEL
LIN {X 0,Y 340.829,Z 506.651,A -85,B 0,C 180,E1 -14238.467,E2 -14238.467} C_VEL
LIN {X 0,Y 340.747,Z 506.663,A -85,B 0,C 180,E1 -14241.858,E2 -14241.858} C_VEL
LIN {X 0,Y 340.766,Z 506.663,A -85,B 0,C 180,E1 -14245.665,E2 -14245.665} C_VEL
LIN {X 0,Y 340.736,Z 506.663,A -85,B 0,C 180,E1 -14248.321,E2 -14248.321} C_VEL
LIN {X 0,Y 340.71,Z 506.668,A -85,B 0,C 180,E1 -14251.044,E2 -14251.044} C_VEL
LIN {X 0,Y 340.714,Z 506.667,A -85,B 0,C 180,E1 -14255.28,E2 -14255.28} C_VEL
LIN {X 0,Y 340.715,Z 506.665,A -85,B 0,C 180,E1 -14258.389,E2 -14258.389} C_VEL
LIN {X 0,Y 340.722,Z 506.668,A -85,B 0,C 180,E1 -14261.305,E2 -14261.305} C_VEL
LIN {X 0,Y 340.778,Z 506.656,A -85,B 0,C 180,E1 -14264.524,E2 -14264.524} C_VEL
LIN {X 0,Y 340.751,Z 506.663,A -85,B 0,C 180,E1 -14267.946,E2 -14267.946} C_VEL
LIN {X 0,Y 340.733,Z 506.664,A -85,B 0,C 180,E1 -14270.254,E2 -14270.254} C_VEL
LIN {X 0,Y 340.71,Z 506.672,A -85,B 0,C 180,E1 -14273.56,E2 -14273.56} C_VEL
LIN {X 0,Y 340.692,Z 506.669,A -85,B 0,C 180,E1 -14276.155,E2 -14276.155} C_VEL
LIN {X 0,Y 340.775,Z 506.659,A -85,B 0,C 180,E1 -14280.334,E2 -14280.334} C_VEL
LIN {X 0,Y 340.806,Z 506.655,A -85,B 0,C 180,E1 -14283.021,E2 -14283.021} C_VEL
LIN {X 0,Y 340.731,Z 506.665,A -85,B 0,C 180,E1 -14286.928,E2 -14286.928} C_VEL
LIN {X 0,Y 340.797,Z 506.654,A -85,B 0,C 180,E1 -14290.735,E2 -14290.735} C_VEL
LIN {X 0,Y 340.79,Z 506.659,A -85,B 0,C 180,E1 -14293.22,E2 -14293.22} C_VEL
LIN {X 0,Y 340.848,Z 506.649,A -85,B 0,C 180,E1 -14296.891,E2 -14296.891} C_VEL
LIN {X 0,Y 340.915,Z 506.64,A -85,B 0,C 180,E1 -14300.508,E2 -14300.508} C_VEL
LIN {X 0,Y 341.051,Z 506.624,A -85,B 0,C 180,E1 -14302.898,E2 -14302.898} C_VEL
LIN {X 0,Y 341.175,Z 506.614,A -85,B 0,C 180,E1 -14307.639,E2 -14307.639} C_VEL
LIN {X 0,Y 341.277,Z 506.598,A -85,B 0,C 180,E1 -14310.001,E2 -14310.001} C_VEL
LIN {X 0,Y 340.934,Z 506.639,A -85,B 0,C 180,E1 -14312.363,E2 -14312.363} C_VEL
LIN {X 0,Y 340.52,Z 506.695,A -85,B 0,C 180,E1 -14315.924,E2 -14315.924} C_VEL
LIN {X 0,Y 340.33,Z 506.89,A -85,B 0,C 180,E1 -14317.591,E2 -14317.591} C_VEL
LIN {X 0,Y 340.122,Z 508.79,A -85,B 0,C 180,E1 -14320.079,E2 -14320.079} C_VEL
LIN {X 0,Y 341.138,Z 511.863,A -85,B 0,C 180,E1 -14320.272,E2 -14320.272} C_VEL
LIN {X 0,Y 346.712,Z 526.262,A -85,B 0,C 180,E1 -14321.288,E2 -14321.288} C_VEL
LIN {X 0,Y 351.362,Z 540.341,A -85,B 0,C 180,E1 -14322.417,E2 -14322.417} C_VEL
LIN {X 0,Y 354.631,Z 552.707,A -85,B 0,C 180,E1 -14323.512,E2 -14323.512} C_VEL
LIN {X 0,Y 353.09,Z 566.451,A -85,B 0,C 180,E1 -14324.554,E2 -14324.554} C_VEL
LIN {X 0,Y 351.191,Z 580.93,A -85,B 0,C 180,E1 -14325.924,E2 -14325.924} C_VEL
LIN {X 0,Y 349.349,Z 593.641,A -85,B 0,C 180,E1 -14327.413,E2 -14327.413} C_VEL
LIN {X 0,Y 347.446,Z 605.162,A -85,B 0,C 180,E1 -14329.037,E2 -14329.037} C_VEL
LIN {X 0,Y 345.461,Z 617.047,A -85,B 0,C 180,E1 -14331.072,E2 -14331.072} C_VEL
LIN {X 0,Y 343.847,Z 626.792,A -85,B 0,C 180,E1 -14333.106,E2 -14333.106} C_VEL
LIN {X 0,Y 342.31,Z 635.783,A -85,B 0,C 180,E1 -14335.394,E2 -14335.394} C_VEL
LIN {X 0,Y 341.201,Z 643.004,A -85,B 0,C 180,E1 -14337.66,E2 -14337.66} C_VEL
LIN {X 0,Y 340.396,Z 648.666,A -85,B 0,C 180,E1 -14339.869,E2 -14339.869} C_VEL
LIN {X 0,Y 339.87,Z 652.973,A -85,B 0,C 180,E1 -14342.024,E2 -14342.024} C_VEL
LIN {X 0,Y 339.417,Z 656.143,A -85,B 0,C 180,E1 -14344.08,E2 -14344.08} C_VEL
LIN {X 0,Y 339.128,Z 658.348,A -85,B 0,C 180,E1 -14346.076,E2 -14346.076} C_VEL
LIN {X 0,Y 338.993,Z 659.888,A -85,B 0,C 180,E1 -14348.459,E2 -14348.459} C_VEL
LIN {X 0,Y 338.98,Z 660.294,A -85,B 0,C 180,E1 -14349.995,E2 -14349.995} C_VEL
LIN {X 0,Y 339,Z 660.201,A -85,B 0,C 180,E1 -14351.725,E2 -14351.725} C_VEL
LIN {X 0,Y 339.14,Z 659.424,A -85,B 0,C 180,E1 -14353.505,E2 -14353.505} C_VEL
LIN {X 0,Y 339.389,Z 658.085,A -85,B 0,C 180,E1 -14355.245,E2 -14355.245} C_VEL
LIN {X 0,Y 339.692,Z 656.205,A -85,B 0,C 180,E1 -14356.94,E2 -14356.94} C_VEL
LIN {X 0,Y 340,Z 654.314,A -85,B 0,C 180,E1 -14358.236,E2 -14358.236} C_VEL
LIN {X 0,Y 339.57,Z 652.788,A -85,B 0,C 180,E1 -14359.193,E2 -14359.193} C_VEL
LIN {X 0,Y 337.21,Z 650.122,A -85,B 0,C 180,E1 -14360.76,E2 -14360.76} C_VEL
LIN {X 0,Y 335.309,Z 647.683,A -85,B 0,C 180,E1 -14362.01,E2 -14362.01} C_VEL
LIN {X 0,Y 334.734,Z 645.517,A -85,B 0,C 180,E1 -14362.95,E2 -14362.95} C_VEL
LIN {X 0,Y 334.818,Z 644.728,A -85,B 0,C 180,E1 -14363.261,E2 -14363.261} C_VEL
LIN {X 0,Y 336.293,Z 637.585,A -85,B 0,C 180,E1 -14365.649,E2 -14365.649} C_VEL
LIN {X 0,Y 337.956,Z 629.452,A -85,B 0,C 180,E1 -14367.848,E2 -14367.848} C_VEL
LIN {X 0,Y 339.959,Z 620.141,A -85,B 0,C 180,E1 -14369.913,E2 -14369.913} C_VEL
LIN {X 0,Y 342.053,Z 609.893,A -85,B 0,C 180,E1 -14371.798,E2 -14371.798} C_VEL
LIN {X 0,Y 344.184,Z 599.122,A -85,B 0,C 180,E1 -14373.451,E2 -14373.451} C_VEL
LIN {X 0,Y 346.355,Z 587.033,A -85,B 0,C 180,E1 -14375,E2 -14375} C_VEL
LIN {X 0,Y 348.444,Z 574.054,A -85,B 0,C 180,E1 -14376.367,E2 -14376.367} C_VEL
LIN {X 0,Y 350.436,Z 560.277,A -85,B 0,C 180,E1 -14377.531,E2 -14377.531} C_VEL
LIN {X 0,Y 350.798,Z 557.022,A -85,B 0,C 180,E1 -14377.78,E2 -14377.78} C_VEL
LIN {X 0,Y 347.291,Z 544.579,A -85,B 0,C 180,E1 -14379.103,E2 -14379.103} C_VEL
LIN {X 0,Y 342.883,Z 532.616,A -85,B 0,C 180,E1 -14380.349,E2 -14380.349} C_VEL
LIN {X 0,Y 338.356,Z 522.719,A -85,B 0,C 180,E1 -14381.379,E2 -14381.379} C_VEL
LIN {X 0,Y 335.067,Z 516.203,A -85,B 0,C 180,E1 -14382.057,E2 -14382.057} C_VEL
LIN {X 0,Y 333.729,Z 513.271,A -85,B 0,C 180,E1 -14382.339,E2 -14382.339} C_VEL
LIN {X 0,Y 333.62,Z 512.653,A -85,B 0,C 180,E1 -14382.412,E2 -14382.412} C_VEL
LIN {X 0,Y 333.833,Z 510.839,A -85,B 0,C 180,E1 -14385.559,E2 -14385.559} C_VEL
LIN {X 0,Y 333.933,Z 508.971,A -85,B 0,C 180,E1 -14389.081,E2 -14389.081} C_VEL
LIN {X 0,Y 333.977,Z 507.76,A -85,B 0,C 180,E1 -14391.529,E2 -14391.529} C_VEL
LIN {X 0,Y 334.014,Z 507.505,A -85,B 0,C 180,E1 -14393.961,E2 -14393.961} C_VEL
LIN {X 0,Y 334.105,Z 507.495,A -85,B 0,C 180,E1 -14397.588,E2 -14397.588} C_VEL
LIN {X 0,Y 334.245,Z 507.475,A -85,B 0,C 180,E1 -14400,E2 -14400} C_VEL
LIN {X 0,Y 334.105,Z 507.494,A -85,B 0,C 180,E1 -14402.411,E2 -14402.411} C_VEL
LIN {X 0,Y 334.023,Z 507.501,A -85,B 0,C 180,E1 -14407.252,E2 -14407.252} C_VEL
LIN {X 0,Y 333.831,Z 507.525,A -85,B 0,C 180,E1 -14410.922,E2 -14410.922} C_VEL
LIN {X 0,Y 333.806,Z 507.53,A -85,B 0,C 180,E1 -14414.634,E2 -14414.634} C_VEL
LIN {X 0,Y 333.794,Z 507.532,A -85,B 0,C 180,E1 -14418.655,E2 -14418.655} C_VEL
LIN {X 0,Y 333.69,Z 507.547,A -85,B 0,C 180,E1 -14422.278,E2 -14422.278} C_VEL
LIN {X 0,Y 333.733,Z 507.539,A -85,B 0,C 180,E1 -14426.246,E2 -14426.246} C_VEL
LIN {X 0,Y 333.709,Z 507.543,A -85,B 0,C 180,E1 -14428.972,E2 -14428.972} C_VEL
LIN {X 0,Y 333.766,Z 508.007,A -85,B 0,C 180,E1 -14430.355,E2 -14430.355} C_VEL
LIN {X 0,Y 334.32,Z 511.125,A -85,B 0,C 180,E1 -14434.582,E2 -14434.582} C_VEL
LIN {X 0,Y 334.755,Z 513.721,A -85,B 0,C 180,E1 -14437.505,E2 -14437.505} C_VEL
LIN {X 0,Y 335.393,Z 517.271,A -85,B 0,C 180,E1 -14441.031,E2 -14441.031} C_VEL
LIN {X 0,Y 336.189,Z 522.177,A -85,B 0,C 180,E1 -14445.297,E2 -14445.297} C_VEL
LIN {X 0,Y 336.39,Z 524.345,A -85,B 0,C 180,E1 -14446.99,E2 -14446.99} C_VEL
LIN {X 0,Y 336.081,Z 527.98,A -85,B 0,C 180,E1 -14449.59,E2 -14449.59} C_VEL
LIN {X 0,Y 335.417,Z 532.753,A -85,B 0,C 180,E1 -14452.77,E2 -14452.77} C_VEL
LIN {X 0,Y 334.747,Z 538.187,A -85,B 0,C 180,E1 -14456.195,E2 -14456.195} C_VEL
LIN {X 0,Y 334.499,Z 540.823,A -85,B 0,C 180,E1 -14457.721,E2 -14457.721} C_VEL
LIN {X 0,Y 335.423,Z 544.098,A -85,B 0,C 180,E1 -14457.941,E2 -14457.941} C_VEL
LIN {X 0,Y 339.831,Z 556.988,A -85,B 0,C 180,E1 -14458.962,E2 -14458.962} C_VEL
LIN {X 0,Y 343.504,Z 570.917,A -85,B 0,C 180,E1 -14460.1,E2 -14460.1} C_VEL
LIN {X 0,Y 346.071,Z 585.53,A -85,B 0,C 180,E1 -14461.348,E2 -14461.348} C_VEL
LIN {X 0,Y 347.375,Z 598.167,A -85,B 0,C 180,E1 -14462.513,E2 -14462.513} C_VEL
LIN {X 0,Y 347.427,Z 603.292,A -85,B 0,C 180,E1 -14463.003,E2 -14463.003} C_VEL
LIN {X 0,Y 345.268,Z 616.264,A -85,B 0,C 180,E1 -14464.209,E2 -14464.209} C_VEL
LIN {X 0,Y 343.018,Z 628.951,A -85,B 0,C 180,E1 -14465.648,E2 -14465.648} C_VEL
LIN {X 0,Y 340.773,Z 640.727,A -85,B 0,C 180,E1 -14467.251,E2 -14467.251} C_VEL
LIN {X 0,Y 338.696,Z 651.614,A -85,B 0,C 180,E1 -14469.028,E2 -14469.028} C_VEL
LIN {X 0,Y 336.746,Z 662.274,A -85,B 0,C 180,E1 -14471.126,E2 -14471.126} C_VEL
LIN {X 0,Y 335.097,Z 671.206,A -85,B 0,C 180,E1 -14473.239,E2 -14473.239} C_VEL
LIN {X 0,Y 333.861,Z 678.699,A -85,B 0,C 180,E1 -14475.368,E2 -14475.368} C_VEL
LIN {X 0,Y 332.955,Z 685.707,A -85,B 0,C 180,E1 -14477.814,E2 -14477.814} C_VEL
LIN {X 0,Y 332.349,Z 691.251,A -85,B 0,C 180,E1 -14480.26,E2 -14480.26} C_VEL
LIN {X 0,Y 332.144,Z 695.431,A -85,B 0,C 180,E1 -14482.706,E2 -14482.706} C_VEL
LIN {X 0,Y 332.075,Z 698.342,A -85,B 0,C 180,E1 -14485.143,E2 -14485.143} C_VEL
LIN {X 0,Y 332.098,Z 700.053,A -85,B 0,C 180,E1 -14487.574,E2 -14487.574} C_VEL
LIN {X 0,Y 332.275,Z 700.595,A -85,B 0,C 180,E1 -14489.999,E2 -14489.999} C_VEL
LIN {X 0,Y 332.103,Z 699.937,A -85,B 0,C 180,E1 -14492.425,E2 -14492.425} C_VEL
LIN {X 0,Y 332.104,Z 698.046,A -85,B 0,C 180,E1 -14494.855,E2 -14494.855} C_VEL
LIN {X 0,Y 332.159,Z 694.909,A -85,B 0,C 180,E1 -14497.293,E2 -14497.293} C_VEL
LIN {X 0,Y 332.351,Z 690.47,A -85,B 0,C 180,E1 -14499.739,E2 -14499.739} C_VEL
LIN {X 0,Y 332.934,Z 684.628,A -85,B 0,C 180,E1 -14502.186,E2 -14502.186} C_VEL
LIN {X 0,Y 333.807,Z 677.221,A -85,B 0,C 180,E1 -14504.633,E2 -14504.633} C_VEL
LIN {X 0,Y 334.993,Z 669.293,A -85,B 0,C 180,E1 -14506.765,E2 -14506.765} C_VEL
LIN {X 0,Y 336.617,Z 659.773,A -85,B 0,C 180,E1 -14508.881,E2 -14508.881} C_VEL
LIN {X 0,Y 338.485,Z 648.455,A -85,B 0,C 180,E1 -14510.954,E2 -14510.954} C_VEL
LIN {X 0,Y 340.463,Z 636.421,A -85,B 0,C 180,E1 -14512.77,E2 -14512.77} C_VEL
LIN {X 0,Y 342.363,Z 624.661,A -85,B 0,C 180,E1 -14514.239,E2 -14514.239} C_VEL
LIN {X 0,Y 344.572,Z 610.894,A -85,B 0,C 180,E1 -14515.64,E2 -14515.64} C_VEL
LIN {X 0,Y 345.847,Z 600.299,A -85,B 0,C 180,E1 -14516.554,E2 -14516.554} C_VEL
LIN {X 0,Y 343.825,Z 585.203,A -85,B 0,C 180,E1 -14517.866,E2 -14517.866} C_VEL
LIN {X 0,Y 340.884,Z 569.74,A -85,B 0,C 180,E1 -14519.021,E2 -14519.021} C_VEL
LIN {X 0,Y 336.796,Z 553.481,A -85,B 0,C 180,E1 -14520.053,E2 -14520.053} C_VEL
LIN {X 0,Y 334.186,Z 543.915,A -85,B 0,C 180,E1 -14520.6,E2 -14520.6} C_VEL
LIN {X 0,Y 334.793,Z 538.415,A -85,B 0,C 180,E1 -14523.798,E2 -14523.798} C_VEL
LIN {X 0,Y 335.455,Z 532.455,A -85,B 0,C 180,E1 -14527.412,E2 -14527.412} C_VEL
LIN {X 0,Y 336.168,Z 527.651,A -85,B 0,C 180,E1 -14530.396,E2 -14530.396} C_VEL
LIN {X 0,Y 336.423,Z 523.629,A -85,B 0,C 180,E1 -14533.016,E2 -14533.016} C_VEL
LIN {X 0,Y 336.015,Z 520.317,A -85,B 0,C 180,E1 -14535.325,E2 -14535.325} C_VEL
LIN {X 0,Y 334.926,Z 514.824,A -85,B 0,C 180,E1 -14539.422,E2 -14539.422} C_VEL
LIN {X 0,Y 334.156,Z 510.27,A -85,B 0,C 180,E1 -14543.053,E2 -14543.053} C_VEL
LIN {X 0,Y 333.673,Z 507.546,A -85,B 0,C 180,E1 -14545.525,E2 -14545.525} C_VEL
LIN {X 0,Y 333.694,Z 507.544,A -85,B 0,C 180,E1 -14549.71,E2 -14549.71} C_VEL
LIN {X 0,Y 333.736,Z 507.536,A -85,B 0,C 180,E1 -14552.401,E2 -14552.401} C_VEL
LIN {X 0,Y 333.717,Z 507.54,A -85,B 0,C 180,E1 -14555.09,E2 -14555.09} C_VEL
LIN {X 0,Y 333.666,Z 507.546,A -85,B 0,C 180,E1 -14559.019,E2 -14559.019} C_VEL
LIN {X 0,Y 333.785,Z 507.535,A -85,B 0,C 180,E1 -14561.589,E2 -14561.589} C_VEL
LIN {X 0,Y 333.799,Z 507.533,A -85,B 0,C 180,E1 -14565.577,E2 -14565.577} C_VEL
LIN {X 0,Y 333.828,Z 507.525,A -85,B 0,C 180,E1 -14569.078,E2 -14569.078} C_VEL
LIN {X 0,Y 334.016,Z 507.499,A -85,B 0,C 180,E1 -14572.748,E2 -14572.748} C_VEL
LIN {X 0,Y 333.807,Z 507.529,A -85,B 0,C 180,E1 -14575.169,E2 -14575.169} C_VEL
LIN {X 0,Y 334.123,Z 507.491,A -85,B 0,C 180,E1 -14577.589,E2 -14577.589} C_VEL
LIN {X 0,Y 334.239,Z 507.47,A -85,B 0,C 180,E1 -14580,E2 -14580} C_VEL
LIN {X 0,Y 334.1,Z 507.487,A -85,B 0,C 180,E1 -14582.412,E2 -14582.412} C_VEL
LIN {X 0,Y 333.988,Z 507.504,A -85,B 0,C 180,E1 -14586.596,E2 -14586.596} C_VEL
LIN {X 0,Y 333.842,Z 507.524,A -85,B 0,C 180,E1 -14589.696,E2 -14589.696} C_VEL
LIN {X 0,Y 333.788,Z 507.528,A -85,B 0,C 180,E1 -14593.392,E2 -14593.392} C_VEL
LIN {X 0,Y 333.738,Z 507.536,A -85,B 0,C 180,E1 -14597.147,E2 -14597.147} C_VEL
LIN {X 0,Y 333.729,Z 507.54,A -85,B 0,C 180,E1 -14599.691,E2 -14599.691} C_VEL
LIN {X 0,Y 333.685,Z 507.539,A -85,B 0,C 180,E1 -14602.279,E2 -14602.279} C_VEL
LIN {X 0,Y 333.729,Z 507.535,A -85,B 0,C 180,E1 -14606.247,E2 -14606.247} C_VEL
LIN {X 0,Y 333.706,Z 507.54,A -85,B 0,C 180,E1 -14608.973,E2 -14608.973} C_VEL
LIN {X 0,Y 333.646,Z 507.545,A -85,B 0,C 180,E1 -14612.59,E2 -14612.59} C_VEL
LIN {X 0,Y 333.673,Z 507.541,A -85,B 0,C 180,E1 -14616.14,E2 -14616.14} C_VEL
LIN {X 0,Y 333.681,Z 507.543,A -85,B 0,C 180,E1 -14619.188,E2 -14619.188} C_VEL
LIN {X 0,Y 333.7,Z 507.539,A -85,B 0,C 180,E1 -14622.515,E2 -14622.515} C_VEL
LIN {X 0,Y 333.726,Z 507.535,A -85,B 0,C 180,E1 -14625.978,E2 -14625.978} C_VEL
LIN {X 0,Y 333.7,Z 507.542,A -85,B 0,C 180,E1 -14629.306,E2 -14629.306} C_VEL
LIN {X 0,Y 333.665,Z 507.546,A -85,B 0,C 180,E1 -14633.169,E2 -14633.169} C_VEL
LIN {X 0,Y 333.674,Z 507.545,A -85,B 0,C 180,E1 -14635.343,E2 -14635.343} C_VEL
LIN {X 0,Y 333.703,Z 507.545,A -85,B 0,C 180,E1 -14639.712,E2 -14639.712} C_VEL
LIN {X 0,Y 333.744,Z 507.533,A -85,B 0,C 180,E1 -14642.403,E2 -14642.403} C_VEL
LIN {X 0,Y 333.728,Z 507.536,A -85,B 0,C 180,E1 -14645.092,E2 -14645.092} C_VEL
LIN {X 0,Y 333.684,Z 507.542,A -85,B 0,C 180,E1 -14649.021,E2 -14649.021} C_VEL
LIN {X 0,Y 333.797,Z 507.532,A -85,B 0,C 180,E1 -14651.591,E2 -14651.591} C_VEL
LIN {X 0,Y 333.812,Z 507.53,A -85,B 0,C 180,E1 -14655.578,E2 -14655.578} C_VEL
LIN {X 0,Y 333.837,Z 507.524,A -85,B 0,C 180,E1 -14659.079,E2 -14659.079} C_VEL
LIN {X 0,Y 333.998,Z 507.503,A -85,B 0,C 180,E1 -14662.748,E2 -14662.748} C_VEL
LIN {X 0,Y 333.814,Z 507.526,A -85,B 0,C 180,E1 -14665.17,E2 -14665.17} C_VEL
LIN {X 0,Y 334.112,Z 507.493,A -85,B 0,C 180,E1 -14667.59,E2 -14667.59} C_VEL
LIN {X 0,Y 334.228,Z 507.476,A -85,B 0,C 180,E1 -14670.001,E2 -14670.001} C_VEL
LIN {X 0,Y 333.885,Z 507.518,A -85,B 0,C 180,E1 -14672.413,E2 -14672.413} C_VEL
LIN {X 0,Y 333.465,Z 507.573,A -85,B 0,C 180,E1 -14676.049,E2 -14676.049} C_VEL
LIN {X 0,Y 333.287,Z 507.824,A -85,B 0,C 180,E1 -14677.65,E2 -14677.65} C_VEL
LIN {X 0,Y 333.132,Z 509.163,A -85,B 0,C 180,E1 -14679.449,E2 -14679.449} C_VEL
LIN {X 0,Y 334.082,Z 512.189,A -85,B 0,C 180,E1 -14679.651,E2 -14679.651} C_VEL
LIN {X 0,Y 340.076,Z 527.413,A -85,B 0,C 180,E1 -14680.776,E2 -14680.776} C_VEL
LIN {X 0,Y 344.59,Z 541.275,A -85,B 0,C 180,E1 -14681.919,E2 -14681.919} C_VEL
LIN {X 0,Y 347.826,Z 553.075,A -85,B 0,C 180,E1 -14683.005,E2 -14683.005} C_VEL
LIN {X 0,Y 348.045,Z 554.809,A -85,B 0,C 180,E1 -14683.16,E2 -14683.16} C_VEL
LIN {X 0,Y 346.351,Z 568.561,A -85,B 0,C 180,E1 -14684.243,E2 -14684.243} C_VEL
LIN {X 0,Y 344.468,Z 582.288,A -85,B 0,C 180,E1 -14685.597,E2 -14685.597} C_VEL
LIN {X 0,Y 342.524,Z 595.147,A -85,B 0,C 180,E1 -14687.155,E2 -14687.155} C_VEL
LIN {X 0,Y 340.554,Z 606.752,A -85,B 0,C 180,E1 -14688.85,E2 -14688.85} C_VEL
LIN {X 0,Y 338.738,Z 617.056,A -85,B 0,C 180,E1 -14690.653,E2 -14690.653} C_VEL
LIN {X 0,Y 337.098,Z 626.478,A -85,B 0,C 180,E1 -14692.636,E2 -14692.636} C_VEL
LIN {X 0,Y 335.602,Z 634.866,A -85,B 0,C 180,E1 -14694.761,E2 -14694.761} C_VEL
LIN {X 0,Y 334.357,Z 642.727,A -85,B 0,C 180,E1 -14697.205,E2 -14697.205} C_VEL
LIN {X 0,Y 333.401,Z 648.764,A -85,B 0,C 180,E1 -14699.568,E2 -14699.568} C_VEL
LIN {X 0,Y 332.84,Z 653.319,A -85,B 0,C 180,E1 -14701.863,E2 -14701.863} C_VEL
LIN {X 0,Y 332.267,Z 657.073,A -85,B 0,C 180,E1 -14704.419,E2 -14704.419} C_VEL
LIN {X 0,Y 332.011,Z 659.13,A -85,B 0,C 180,E1 -14706.448,E2 -14706.448} C_VEL
LIN {X 0,Y 331.92,Z 660.294,A -85,B 0,C 180,E1 -14708.423,E2 -14708.423} C_VEL
LIN {X 0,Y 331.886,Z 660.724,A -85,B 0,C 180,E1 -14711.03,E2 -14711.03} C_VEL
LIN {X 0,Y 331.979,Z 660.344,A -85,B 0,C 180,E1 -14712.644,E2 -14712.644} C_VEL
LIN {X 0,Y 332.14,Z 659.46,A -85,B 0,C 180,E1 -14714.288,E2 -14714.288} C_VEL
LIN {X 0,Y 332.415,Z 657.992,A -85,B 0,C 180,E1 -14715.958,E2 -14715.958} C_VEL
LIN {X 0,Y 332.992,Z 654.834,A -85,B 0,C 180,E1 -14718.417,E2 -14718.417} C_VEL
LIN {X 0,Y 333.854,Z 649.782,A -85,B 0,C 180,E1 -14721.159,E2 -14721.159} C_VEL
LIN {X 0,Y 334.818,Z 644.728,A -85,B 0,C 180,E1 -14723.261,E2 -14723.261} C_VEL
LIN {X 0,Y 334.707,Z 642.345,A -85,B 0,C 180,E1 -14724.186,E2 -14724.186} C_VEL
LIN {X 0,Y 332.892,Z 638.3,A -85,B 0,C 180,E1 -14725.707,E2 -14725.707} C_VEL
LIN {X 0,Y 331.129,Z 633.811,A -85,B 0,C 180,E1 -14727.204,E2 -14727.204} C_VEL
LIN {X 0,Y 331.097,Z 630.688,A -85,B 0,C 180,E1 -14728.076,E2 -14728.076} C_VEL
LIN {X 0,Y 333.235,Z 621.325,A -85,B 0,C 180,E1 -14730.23,E2 -14730.23} C_VEL
LIN {X 0,Y 335.451,Z 611.04,A -85,B 0,C 180,E1 -14732.188,E2 -14732.188} C_VEL
LIN {X 0,Y 337.759,Z 599.949,A -85,B 0,C 180,E1 -14733.936,E2 -14733.936} C_VEL
LIN {X 0,Y 340.126,Z 587.265,A -85,B 0,C 180,E1 -14735.59,E2 -14735.59} C_VEL
LIN {X 0,Y 342.458,Z 573.448,A -85,B 0,C 180,E1 -14737.05,E2 -14737.05} C_VEL
LIN {X 0,Y 344.375,Z 560.7,A -85,B 0,C 180,E1 -14738.133,E2 -14738.133} C_VEL
LIN {X 0,Y 344.511,Z 558.707,A -85,B 0,C 180,E1 -14738.299,E2 -14738.299} C_VEL
LIN {X 0,Y 340.922,Z 545.95,A -85,B 0,C 180,E1 -14739.732,E2 -14739.732} C_VEL
LIN {X 0,Y 336.091,Z 533.059,A -85,B 0,C 180,E1 -14741.146,E2 -14741.146} C_VEL
LIN {X 0,Y 331.381,Z 523.017,A -85,B 0,C 180,E1 -14742.267,E2 -14742.267} C_VEL
LIN {X 0,Y 328.153,Z 516.855,A -85,B 0,C 180,E1 -14742.953,E2 -14742.953} C_VEL
LIN {X 0,Y 326.815,Z 514.13,A -85,B 0,C 180,E1 -14743.244,E2 -14743.244} C_VEL
LIN {X 0,Y 326.629,Z 513.232,A -85,B 0,C 180,E1 -14743.354,E2 -14743.354} C_VEL
LIN {X 0,Y 326.849,Z 511.591,A -85,B 0,C 180,E1 -14746.318,E2 -14746.318} C_VEL
LIN {X 0,Y 326.949,Z 509.691,A -85,B 0,C 180,E1 -14750.097,E2 -14750.097} C_VEL
LIN {X 0,Y 326.982,Z 508.533,A -85,B 0,C 180,E1 -14752.59,E2 -14752.59} C_VEL
LIN {X 0,Y 326.988,Z 508.381,A -85,B 0,C 180,E1 -14753.83,E2 -14753.83} C_VEL
LIN {X 0,Y 327.046,Z 508.374,A -85,B 0,C 180,E1 -14757.536,E2 -14757.536} C_VEL
LIN {X 0,Y 327.196,Z 508.352,A -85,B 0,C 180,E1 -14760,E2 -14760} C_VEL
LIN {X 0,Y 327.045,Z 508.373,A -85,B 0,C 180,E1 -14762.463,E2 -14762.463} C_VEL
LIN {X 0,Y 326.994,Z 508.379,A -85,B 0,C 180,E1 -14766.169,E2 -14766.169} C_VEL
LIN {X 0,Y 326.913,Z 508.389,A -85,B 0,C 180,E1 -14768.655,E2 -14768.655} C_VEL
LIN {X 0,Y 326.732,Z 508.412,A -85,B 0,C 180,E1 -14772.421,E2 -14772.421} C_VEL
LIN {X 0,Y 326.752,Z 508.406,A -85,B 0,C 180,E1 -14774.957,E2 -14774.957} C_VEL
LIN {X 0,Y 326.73,Z 508.41,A -85,B 0,C 180,E1 -14778.838,E2 -14778.838} C_VEL
LIN {X 0,Y 326.618,Z 508.424,A -85,B 0,C 180,E1 -14782.787,E2 -14782.787} C_VEL
LIN {X 0,Y 326.688,Z 508.416,A -85,B 0,C 180,E1 -14785.483,E2 -14785.483} C_VEL
LIN {X 0,Y 326.655,Z 508.42,A -85,B 0,C 180,E1 -14788.25,E2 -14788.25} C_VEL
LIN {X 0,Y 326.894,Z 510.08,A -85,B 0,C 180,E1 -14791.063,E2 -14791.063} C_VEL
LIN {X 0,Y 327.267,Z 512.182,A -85,B 0,C 180,E1 -14793.941,E2 -14793.941} C_VEL
LIN {X 0,Y 327.812,Z 515.204,A -85,B 0,C 180,E1 -14797.51,E2 -14797.51} C_VEL
LIN {X 0,Y 328.228,Z 517.579,A -85,B 0,C 180,E1 -14799.967,E2 -14799.967} C_VEL
LIN {X 0,Y 328.799,Z 521.27,A -85,B 0,C 180,E1 -14803.386,E2 -14803.386} C_VEL
LIN {X 0,Y 329.403,Z 525,A -85,B 0,C 180,E1 -14806.502,E2 -14806.502} C_VEL
LIN {X 0,Y 329.259,Z 527.737,A -85,B 0,C 180,E1 -14808.571,E2 -14808.571} C_VEL
LIN {X 0,Y 328.493,Z 533.174,A -85,B 0,C 180,E1 -14812.335,E2 -14812.335} C_VEL
LIN {X 0,Y 327.739,Z 539.01,A -85,B 0,C 180,E1 -14816.114,E2 -14816.114} C_VEL
LIN {X 0,Y 327.577,Z 540.109,A -85,B 0,C 180,E1 -14816.795,E2 -14816.795} C_VEL
LIN {X 0,Y 328.449,Z 543.269,A -85,B 0,C 180,E1 -14817.018,E2 -14817.018} C_VEL
LIN {X 0,Y 330.844,Z 549.552,A -85,B 0,C 180,E1 -14817.559,E2 -14817.559} C_VEL
LIN {X 0,Y 335.072,Z 563.283,A -85,B 0,C 180,E1 -14818.727,E2 -14818.727} C_VEL
LIN {X 0,Y 338.203,Z 576.867,A -85,B 0,C 180,E1 -14819.912,E2 -14819.912} C_VEL
LIN {X 0,Y 340.235,Z 590.765,A -85,B 0,C 180,E1 -14821.191,E2 -14821.191} C_VEL
LIN {X 0,Y 341.085,Z 602.706,A -85,B 0,C 180,E1 -14822.375,E2 -14822.375} C_VEL
LIN {X 0,Y 338.87,Z 616.404,A -85,B 0,C 180,E1 -14823.685,E2 -14823.685} C_VEL
LIN {X 0,Y 336.532,Z 628.986,A -85,B 0,C 180,E1 -14825.147,E2 -14825.147} C_VEL
LIN {X 0,Y 334.604,Z 638.686,A -85,B 0,C 180,E1 -14826.479,E2 -14826.479} C_VEL
LIN {X 0,Y 332.267,Z 650.115,A -85,B 0,C 180,E1 -14828.34,E2 -14828.34} C_VEL
LIN {X 0,Y 330.24,Z 660.669,A -85,B 0,C 180,E1 -14830.416,E2 -14830.416} C_VEL
LIN {X 0,Y 328.423,Z 669.799,A -85,B 0,C 180,E1 -14832.567,E2 -14832.567} C_VEL
LIN {X 0,Y 326.922,Z 678.405,A -85,B 0,C 180,E1 -14835.05,E2 -14835.05} C_VEL
LIN {X 0,Y 325.928,Z 685.372,A -85,B 0,C 180,E1 -14837.547,E2 -14837.547} C_VEL
LIN {X 0,Y 325.298,Z 690.888,A -85,B 0,C 180,E1 -14840.047,E2 -14840.047} C_VEL
LIN {X 0,Y 325.048,Z 695.055,A -85,B 0,C 180,E1 -14842.546,E2 -14842.546} C_VEL
LIN {X 0,Y 324.977,Z 697.948,A -85,B 0,C 180,E1 -14845.037,E2 -14845.037} C_VEL
LIN {X 0,Y 325.005,Z 699.637,A -85,B 0,C 180,E1 -14847.521,E2 -14847.521} C_VEL
LIN {X 0,Y 325.216,Z 700.16,A -85,B 0,C 180,E1 -14849.999,E2 -14849.999} C_VEL
LIN {X 0,Y 325.009,Z 699.477,A -85,B 0,C 180,E1 -14852.478,E2 -14852.478} C_VEL
LIN {X 0,Y 325.027,Z 697.575,A -85,B 0,C 180,E1 -14854.961,E2 -14854.961} C_VEL
LIN {X 0,Y 325.067,Z 694.408,A -85,B 0,C 180,E1 -14857.453,E2 -14857.453} C_VEL
LIN {X 0,Y 325.3,Z 689.94,A -85,B 0,C 180,E1 -14859.952,E2 -14859.952} C_VEL
LIN {X 0,Y 325.888,Z 684.063,A -85,B 0,C 180,E1 -14862.453,E2 -14862.453} C_VEL
LIN {X 0,Y 326.857,Z 676.623,A -85,B 0,C 180,E1 -14864.952,E2 -14864.952} C_VEL
LIN {X 0,Y 328.093,Z 668.653,A -85,B 0,C 180,E1 -14867.129,E2 -14867.129} C_VEL
LIN {X 0,Y 329.829,Z 659.091,A -85,B 0,C 180,E1 -14869.284,E2 -14869.284} C_VEL
LIN {X 0,Y 331.469,Z 649.336,A -85,B 0,C 180,E1 -14871.126,E2 -14871.126} C_VEL
LIN {X 0,Y 333.465,Z 637.775,A -85,B 0,C 180,E1 -14872.947,E2 -14872.947} C_VEL
LIN {X 0,Y 335.449,Z 626.383,A -85,B 0,C 180,E1 -14874.442,E2 -14874.442} C_VEL
LIN {X 0,Y 337.456,Z 614.177,A -85,B 0,C 180,E1 -14875.768,E2 -14875.768} C_VEL
LIN {X 0,Y 339.153,Z 602.128,A -85,B 0,C 180,E1 -14876.852,E2 -14876.852} C_VEL
LIN {X 0,Y 337.538,Z 588.518,A -85,B 0,C 180,E1 -14878.098,E2 -14878.098} C_VEL
LIN {X 0,Y 334.797,Z 573.068,A -85,B 0,C 180,E1 -14879.324,E2 -14879.324} C_VEL
LIN {X 0,Y 331.018,Z 557.39,A -85,B 0,C 180,E1 -14880.4,E2 -14880.4} C_VEL
LIN {X 0,Y 327.279,Z 543.947,A -85,B 0,C 180,E1 -14881.187,E2 -14881.187} C_VEL
LIN {X 0,Y 327.23,Z 543.564,A -85,B 0,C 180,E1 -14881.206,E2 -14881.206} C_VEL
LIN {X 0,Y 327.912,Z 537.936,A -85,B 0,C 180,E1 -14884.607,E2 -14884.607} C_VEL
LIN {X 0,Y 328.834,Z 530.832,A -85,B 0,C 180,E1 -14889.022,E2 -14889.022} C_VEL
LIN {X 0,Y 329.344,Z 526.729,A -85,B 0,C 180,E1 -14891.68,E2 -14891.68} C_VEL
LIN {X 0,Y 329.365,Z 524.052,A -85,B 0,C 180,E1 -14893.491,E2 -14893.491} C_VEL
LIN {X 0,Y 329.068,Z 521.682,A -85,B 0,C 180,E1 -14895.188,E2 -14895.188} C_VEL
LIN {X 0,Y 328.163,Z 517.223,A -85,B 0,C 180,E1 -14898.551,E2 -14898.551} C_VEL
LIN {X 0,Y 327.27,Z 512.176,A -85,B 0,C 180,E1 -14902.611,E2 -14902.611} C_VEL
LIN {X 0,Y 326.633,Z 508.421,A -85,B 0,C 180,E1 -14905.984,E2 -14905.984} C_VEL
LIN {X 0,Y 326.652,Z 508.417,A -85,B 0,C 180,E1 -14910.341,E2 -14910.341} C_VEL
LIN {X 0,Y 326.681,Z 508.414,A -85,B 0,C 180,E1 -14914.516,E2 -14914.516} C_VEL
LIN {X 0,Y 326.611,Z 508.423,A -85,B 0,C 180,E1 -14918.543,E2 -14918.543} C_VEL
LIN {X 0,Y 326.736,Z 508.41,A -85,B 0,C 180,E1 -14921.177,E2 -14921.177} C_VEL
LIN {X 0,Y 326.754,Z 508.41,A -85,B 0,C 180,E1 -14925.433,E2 -14925.433} C_VEL
LIN {X 0,Y 326.764,Z 508.403,A -85,B 0,C 180,E1 -14928.839,E2 -14928.839} C_VEL
LIN {X 0,Y 326.97,Z 508.376,A -85,B 0,C 180,E1 -14932.591,E2 -14932.591} C_VEL
LIN {X 0,Y 326.773,Z 508.404,A -85,B 0,C 180,E1 -14935.065,E2 -14935.065} C_VEL
LIN {X 0,Y 327.06,Z 508.371,A -85,B 0,C 180,E1 -14937.537,E2 -14937.537} C_VEL
LIN {X 0,Y 327.191,Z 508.347,A -85,B 0,C 180,E1 -14940,E2 -14940} C_VEL
LIN {X 0,Y 327.041,Z 508.366,A -85,B 0,C 180,E1 -14942.464,E2 -14942.464} C_VEL
LIN {X 0,Y 326.957,Z 508.38,A -85,B 0,C 180,E1 -14946.586,E2 -14946.586} C_VEL
LIN {X 0,Y 326.797,Z 508.398,A -85,B 0,C 180,E1 -14949.907,E2 -14949.907} C_VEL
LIN {X 0,Y 326.751,Z 508.407,A -85,B 0,C 180,E1 -14953.686,E2 -14953.686} C_VEL
LIN {X 0,Y 326.692,Z 508.418,A -85,B 0,C 180,E1 -14957.529,E2 -14957.529} C_VEL
LIN {X 0,Y 326.655,Z 508.417,A -85,B 0,C 180,E1 -14960.136,E2 -14960.136} C_VEL
LIN {X 0,Y 326.645,Z 508.414,A -85,B 0,C 180,E1 -14964.13,E2 -14964.13} C_VEL
LIN {X 0,Y 326.679,Z 508.412,A -85,B 0,C 180,E1 -14966.859,E2 -14966.859} C_VEL
LIN {X 0,Y 326.636,Z 508.419,A -85,B 0,C 180,E1 -14970.613,E2 -14970.613} C_VEL
LIN {X 0,Y 326.604,Z 508.421,A -85,B 0,C 180,E1 -14974.02,E2 -14974.02} C_VEL
LIN {X 0,Y 326.627,Z 508.419,A -85,B 0,C 180,E1 -14977.241,E2 -14977.241} C_VEL
LIN {X 0,Y 326.632,Z 508.421,A -85,B 0,C 180,E1 -14980.204,E2 -14980.204} C_VEL
LIN {X 0,Y 326.655,Z 508.422,A -85,B 0,C 180,E1 -14983.511,E2 -14983.511} C_VEL
LIN {X 0,Y 326.649,Z 508.415,A -85,B 0,C 180,E1 -14987.015,E2 -14987.015} C_VEL
LIN {X 0,Y 326.644,Z 508.42,A -85,B 0,C 180,E1 -14990.767,E2 -14990.767} C_VEL
LIN {X 0,Y 326.612,Z 508.421,A -85,B 0,C 180,E1 -14994.482,E2 -14994.482} C_VEL
LIN {X 0,Y 326.607,Z 508.426,A -85,B 0,C 180,E1 -14997.457,E2 -14997.457} C_VEL
LIN {X 0,Y 326.661,Z 508.418,A -85,B 0,C 180,E1 -15000.342,E2 -15000.342} C_VEL
LIN {X 0,Y 326.692,Z 508.411,A -85,B 0,C 180,E1 -15004.518,E2 -15004.518} C_VEL
LIN {X 0,Y 326.649,Z 508.418,A -85,B 0,C 180,E1 -15008.547,E2 -15008.547} C_VEL
LIN {X 0,Y 326.747,Z 508.406,A -85,B 0,C 180,E1 -15011.179,E2 -15011.179} C_VEL
LIN {X 0,Y 326.766,Z 508.407,A -85,B 0,C 180,E1 -15015.434,E2 -15015.434} C_VEL
LIN {X 0,Y 326.773,Z 508.403,A -85,B 0,C 180,E1 -15018.84,E2 -15018.84} C_VEL
LIN {X 0,Y 326.947,Z 508.381,A -85,B 0,C 180,E1 -15022.59,E2 -15022.59} C_VEL
LIN {X 0,Y 326.989,Z 508.378,A -85,B 0,C 180,E1 -15023.832,E2 -15023.832} C_VEL
LIN {X 0,Y 327.053,Z 508.372,A -85,B 0,C 180,E1 -15027.537,E2 -15027.537} C_VEL
LIN {X 0,Y 327.179,Z 508.354,A -85,B 0,C 180,E1 -15030.001,E2 -15030.001} C_VEL
LIN {X 0,Y 326.838,Z 508.396,A -85,B 0,C 180,E1 -15032.465,E2 -15032.465} C_VEL
LIN {X 0,Y 326.412,Z 508.452,A -85,B 0,C 180,E1 -15036.181,E2 -15036.181} C_VEL
LIN {X 0,Y 326.239,Z 508.788,A -85,B 0,C 180,E1 -15037.707,E2 -15037.707} C_VEL
LIN {X 0,Y 326.114,Z 509.605,A -85,B 0,C 180,E1 -15038.803,E2 -15038.803} C_VEL
LIN {X 0,Y 327.253,Z 512.867,A -85,B 0,C 180,E1 -15039.033,E2 -15039.033} C_VEL
LIN {X 0,Y 333.311,Z 528.405,A -85,B 0,C 180,E1 -15040.226,E2 -15040.226} C_VEL
LIN {X 0,Y 337.936,Z 542.584,A -85,B 0,C 180,E1 -15041.444,E2 -15041.444} C_VEL
LIN {X 0,Y 341.51,Z 556.078,A -85,B 0,C 180,E1 -15042.734,E2 -15042.734} C_VEL
LIN {X 0,Y 339.798,Z 569.432,A -85,B 0,C 180,E1 -15043.815,E2 -15043.815} C_VEL
LIN {X 0,Y 337.812,Z 583.379,A -85,B 0,C 180,E1 -15045.228,E2 -15045.228} C_VEL
LIN {X 0,Y 335.823,Z 595.972,A -85,B 0,C 180,E1 -15046.793,E2 -15046.793} C_VEL
LIN {X 0,Y 333.693,Z 607.982,A -85,B 0,C 180,E1 -15048.6,E2 -15048.6} C_VEL
LIN {X 0,Y 331.819,Z 618.235,A -85,B 0,C 180,E1 -15050.455,E2 -15050.455} C_VEL
LIN {X 0,Y 330.095,Z 627.784,A -85,B 0,C 180,E1 -15052.534,E2 -15052.534} C_VEL
LIN {X 0,Y 328.582,Z 635.872,A -85,B 0,C 180,E1 -15054.651,E2 -15054.651} C_VEL
LIN {X 0,Y 327.453,Z 642.582,A -85,B 0,C 180,E1 -15056.79,E2 -15056.79} C_VEL
LIN {X 0,Y 326.516,Z 648.194,A -85,B 0,C 180,E1 -15058.966,E2 -15058.966} C_VEL
LIN {X 0,Y 325.91,Z 652.755,A -85,B 0,C 180,E1 -15061.168,E2 -15061.168} C_VEL
LIN {X 0,Y 325.378,Z 656.349,A -85,B 0,C 180,E1 -15063.421,E2 -15063.421} C_VEL
LIN {X 0,Y 324.998,Z 658.938,A -85,B 0,C 180,E1 -15065.723,E2 -15065.723} C_VEL
LIN {X 0,Y 324.851,Z 660.143,A -85,B 0,C 180,E1 -15067.284,E2 -15067.284} C_VEL
LIN {X 0,Y 324.81,Z 660.907,A -85,B 0,C 180,E1 -15068.864,E2 -15068.864} C_VEL
LIN {X 0,Y 324.796,Z 661.186,A -85,B 0,C 180,E1 -15070.769,E2 -15070.769} C_VEL
LIN {X 0,Y 324.909,Z 660.81,A -85,B 0,C 180,E1 -15072.655,E2 -15072.655} C_VEL
LIN {X 0,Y 325.084,Z 659.865,A -85,B 0,C 180,E1 -15074.485,E2 -15074.485} C_VEL
LIN {X 0,Y 325.615,Z 657.244,A -85,B 0,C 180,E1 -15077.21,E2 -15077.21} C_VEL
LIN {X 0,Y 326.318,Z 653.484,A -85,B 0,C 180,E1 -15079.75,E2 -15079.75} C_VEL
LIN {X 0,Y 327.165,Z 648.898,A -85,B 0,C 180,E1 -15082.059,E2 -15082.059} C_VEL
LIN {X 0,Y 328.416,Z 642.973,A -85,B 0,C 180,E1 -15084.408,E2 -15084.408} C_VEL
LIN {X 0,Y 330.056,Z 635.602,A -85,B 0,C 180,E1 -15086.749,E2 -15086.749} C_VEL
LIN {X 0,Y 331.097,Z 630.688,A -85,B 0,C 180,E1 -15088.076,E2 -15088.076} C_VEL
LIN {X 0,Y 331.145,Z 627.476,A -85,B 0,C 180,E1 -15088.935,E2 -15088.935} C_VEL
LIN {X 0,Y 329.79,Z 622.165,A -85,B 0,C 180,E1 -15090.37,E2 -15090.37} C_VEL
LIN {X 0,Y 328.564,Z 616.438,A -85,B 0,C 180,E1 -15091.758,E2 -15091.758} C_VEL
LIN {X 0,Y 328.791,Z 612.549,A -85,B 0,C 180,E1 -15092.53,E2 -15092.53} C_VEL
LIN {X 0,Y 331.283,Z 601.118,A -85,B 0,C 180,E1 -15094.389,E2 -15094.389} C_VEL
LIN {X 0,Y 333.795,Z 588.423,A -85,B 0,C 180,E1 -15096.093,E2 -15096.093} C_VEL
LIN {X 0,Y 336.135,Z 575.226,A -85,B 0,C 180,E1 -15097.537,E2 -15097.537} C_VEL
LIN {X 0,Y 338.22,Z 562.301,A -85,B 0,C 180,E1 -15098.676,E2 -15098.676} C_VEL
LIN {X 0,Y 338.255,Z 560.523,A -85,B 0,C 180,E1 -15098.838,E2 -15098.838} C_VEL
LIN {X 0,Y 334.976,Z 548.66,A -85,B 0,C 180,E1 -15100.238,E2 -15100.238} C_VEL
LIN {X 0,Y 330.507,Z 536.247,A -85,B 0,C 180,E1 -15101.683,E2 -15101.683} C_VEL
LIN {X 0,Y 325.02,Z 524.475,A -85,B 0,C 180,E1 -15103.067,E2 -15103.067} C_VEL
LIN {X 0,Y 321.321,Z 517.597,A -85,B 0,C 180,E1 -15103.906,E2 -15103.906} C_VEL
LIN {X 0,Y 319.989,Z 515.151,A -85,B 0,C 180,E1 -15104.204,E2 -15104.204} C_VEL
LIN {X 0,Y 319.702,Z 513.83,A -85,B 0,C 180,E1 -15104.336,E2 -15104.336} C_VEL
LIN {X 0,Y 319.881,Z 512.274,A -85,B 0,C 180,E1 -15107.308,E2 -15107.308} C_VEL
LIN {X 0,Y 320.016,Z 510.41,A -85,B 0,C 180,E1 -15111.211,E2 -15111.211} C_VEL
LIN {X 0,Y 319.965,Z 509.357,A -85,B 0,C 180,E1 -15113.694,E2 -15113.694} C_VEL
LIN {X 0,Y 319.99,Z 509.253,A -85,B 0,C 180,E1 -15117.482,E2 -15117.482} C_VEL
LIN {X 0,Y 320.148,Z 509.23,A -85,B 0,C 180,E1 -15120,E2 -15120} C_VEL
LIN {X 0,Y 319.989,Z 509.252,A -85,B 0,C 180,E1 -15122.517,E2 -15122.517} C_VEL
LIN {X 0,Y 319.95,Z 509.257,A -85,B 0,C 180,E1 -15126.305,E2 -15126.305} C_VEL
LIN {X 0,Y 319.84,Z 509.268,A -85,B 0,C 180,E1 -15128.848,E2 -15128.848} C_VEL
LIN {X 0,Y 319.679,Z 509.289,A -85,B 0,C 180,E1 -15132.699,E2 -15132.699} C_VEL
LIN {X 0,Y 319.697,Z 509.284,A -85,B 0,C 180,E1 -15135.295,E2 -15135.295} C_VEL
LIN {X 0,Y 319.672,Z 509.288,A -85,B 0,C 180,E1 -15139.255,E2 -15139.255} C_VEL
LIN {X 0,Y 319.568,Z 509.301,A -85,B 0,C 180,E1 -15143.319,E2 -15143.319} C_VEL
LIN {X 0,Y 319.633,Z 509.297,A -85,B 0,C 180,E1 -15146.088,E2 -15146.088} C_VEL
LIN {X 0,Y 319.656,Z 509.524,A -85,B 0,C 180,E1 -15147.497,E2 -15147.497} C_VEL
LIN {X 0,Y 319.994,Z 511.674,A -85,B 0,C 180,E1 -15151.069,E2 -15151.069} C_VEL
LIN {X 0,Y 320.451,Z 514.383,A -85,B 0,C 180,E1 -15154.765,E2 -15154.765} C_VEL
LIN {X 0,Y 320.953,Z 517.118,A -85,B 0,C 180,E1 -15157.973,E2 -15157.973} C_VEL
LIN {X 0,Y 321.423,Z 520.067,A -85,B 0,C 180,E1 -15160.992,E2 -15160.992} C_VEL
LIN {X 0,Y 322.005,Z 523.677,A -85,B 0,C 180,E1 -15164.3,E2 -15164.3} C_VEL
LIN {X 0,Y 322.342,Z 525.675,A -85,B 0,C 180,E1 -15166.012,E2 -15166.012} C_VEL
LIN {X 0,Y 322.338,Z 528.001,A -85,B 0,C 180,E1 -15167.843,E2 -15167.843} C_VEL
LIN {X 0,Y 321.808,Z 531.934,A -85,B 0,C 180,E1 -15170.704,E2 -15170.704} C_VEL
LIN {X 0,Y 321.103,Z 536.867,A -85,B 0,C 180,E1 -15174.078,E2 -15174.078} C_VEL
LIN {X 0,Y 320.746,Z 539.519,A -85,B 0,C 180,E1 -15175.817,E2 -15175.817} C_VEL
LIN {X 0,Y 321.76,Z 543.04,A -85,B 0,C 180,E1 -15176.099,E2 -15176.099} C_VEL
LIN {X 0,Y 322.774,Z 545.601,A -85,B 0,C 180,E1 -15176.342,E2 -15176.342} C_VEL
LIN {X 0,Y 327.383,Z 558.869,A -85,B 0,C 180,E1 -15177.542,E2 -15177.542} C_VEL
LIN {X 0,Y 331.296,Z 574.454,A -85,B 0,C 180,E1 -15178.97,E2 -15178.97} C_VEL
LIN {X 0,Y 333.621,Z 589.234,A -85,B 0,C 180,E1 -15180.372,E2 -15180.372} C_VEL
LIN {X 0,Y 334.658,Z 602.728,A -85,B 0,C 180,E1 -15181.764,E2 -15181.764} C_VEL
LIN {X 0,Y 334.324,Z 606.906,A -85,B 0,C 180,E1 -15182.183,E2 -15182.183} C_VEL
LIN {X 0,Y 331.751,Z 620.495,A -85,B 0,C 180,E1 -15183.584,E2 -15183.584} C_VEL
LIN {X 0,Y 329.147,Z 633.446,A -85,B 0,C 180,E1 -15185.226,E2 -15185.226} C_VEL
LIN {X 0,Y 326.809,Z 644.382,A -85,B 0,C 180,E1 -15186.892,E2 -15186.892} C_VEL
LIN {X 0,Y 324.509,Z 655.242,A -85,B 0,C 180,E1 -15188.88,E2 -15188.88} C_VEL
LIN {X 0,Y 322.583,Z 664.578,A -85,B 0,C 180,E1 -15190.925,E2 -15190.925} C_VEL
LIN {X 0,Y 320.753,Z 674.045,A -85,B 0,C 180,E1 -15193.45,E2 -15193.45} C_VEL
LIN {X 0,Y 319.364,Z 681.77,A -85,B 0,C 180,E1 -15195.991,E2 -15195.991} C_VEL
LIN {X 0,Y 318.514,Z 687.965,A -85,B 0,C 180,E1 -15198.545,E2 -15198.545} C_VEL
LIN {X 0,Y 318.074,Z 692.782,A -85,B 0,C 180,E1 -15201.102,E2 -15201.102} C_VEL
LIN {X 0,Y 317.904,Z 696.274,A -85,B 0,C 180,E1 -15203.653,E2 -15203.653} C_VEL
LIN {X 0,Y 317.909,Z 698.538,A -85,B 0,C 180,E1 -15206.197,E2 -15206.197} C_VEL
LIN {X 0,Y 318.048,Z 699.622,A -85,B 0,C 180,E1 -15208.733,E2 -15208.733} C_VEL
LIN {X 0,Y 318.14,Z 699.724,A -85,B 0,C 180,E1 -15209.999,E2 -15209.999} C_VEL
LIN {X 0,Y 317.92,Z 699.017,A -85,B 0,C 180,E1 -15212.533,E2 -15212.533} C_VEL
LIN {X 0,Y 317.935,Z 697.103,A -85,B 0,C 180,E1 -15215.072,E2 -15215.072} C_VEL
LIN {X 0,Y 317.988,Z 693.908,A -85,B 0,C 180,E1 -15217.62,E2 -15217.62} C_VEL
LIN {X 0,Y 318.236,Z 689.409,A -85,B 0,C 180,E1 -15220.175,E2 -15220.175} C_VEL
LIN {X 0,Y 318.857,Z 683.498,A -85,B 0,C 180,E1 -15222.732,E2 -15222.732} C_VEL
LIN {X 0,Y 319.92,Z 676.025,A -85,B 0,C 180,E1 -15225.284,E2 -15225.284} C_VEL
LIN {X 0,Y 321.205,Z 668.014,A -85,B 0,C 180,E1 -15227.508,E2 -15227.508} C_VEL
LIN {X 0,Y 323.043,Z 658.408,A -85,B 0,C 180,E1 -15229.706,E2 -15229.706} C_VEL
LIN {X 0,Y 324.773,Z 648.602,A -85,B 0,C 180,E1 -15231.584,E2 -15231.584} C_VEL
LIN {X 0,Y 326.853,Z 636.969,A -85,B 0,C 180,E1 -15233.439,E2 -15233.439} C_VEL
LIN {X 0,Y 328.866,Z 625.481,A -85,B 0,C 180,E1 -15234.964,E2 -15234.964} C_VEL
LIN {X 0,Y 331.021,Z 613.218,A -85,B 0,C 180,E1 -15236.307,E2 -15236.307} C_VEL
LIN {X 0,Y 332.47,Z 602.819,A -85,B 0,C 180,E1 -15237.264,E2 -15237.264} C_VEL
LIN {X 0,Y 330.79,Z 588.903,A -85,B 0,C 180,E1 -15238.585,E2 -15238.585} C_VEL
LIN {X 0,Y 328.122,Z 573.793,A -85,B 0,C 180,E1 -15239.834,E2 -15239.834} C_VEL
LIN {X 0,Y 324.308,Z 557.708,A -85,B 0,C 180,E1 -15240.986,E2 -15240.986} C_VEL
LIN {X 0,Y 320.319,Z 543.161,A -85,B 0,C 180,E1 -15241.886,E2 -15241.886} C_VEL
LIN {X 0,Y 321.102,Z 536.63,A -85,B 0,C 180,E1 -15245.922,E2 -15245.922} C_VEL
LIN {X 0,Y 322.025,Z 530.007,A -85,B 0,C 180,E1 -15250.195,E2 -15250.195} C_VEL
LIN {X 0,Y 322.397,Z 526.577,A -85,B 0,C 180,E1 -15252.513,E2 -15252.513} C_VEL
LIN {X 0,Y 322.194,Z 524.106,A -85,B 0,C 180,E1 -15254.266,E2 -15254.266} C_VEL
LIN {X 0,Y 321.487,Z 520.019,A -85,B 0,C 180,E1 -15257.337,E2 -15257.337} C_VEL
LIN {X 0,Y 320.75,Z 515.986,A -85,B 0,C 180,E1 -15260.549,E2 -15260.549} C_VEL
LIN {X 0,Y 319.931,Z 511.488,A -85,B 0,C 180,E1 -15264.367,E2 -15264.367} C_VEL
LIN {X 0,Y 319.579,Z 509.3,A -85,B 0,C 180,E1 -15266.459,E2 -15266.459} C_VEL
LIN {X 0,Y 319.583,Z 509.303,A -85,B 0,C 180,E1 -15269.616,E2 -15269.616} C_VEL
LIN {X 0,Y 319.6,Z 509.297,A -85,B 0,C 180,E1 -15272.498,E2 -15272.498} C_VEL
LIN {X 0,Y 319.594,Z 509.301,A -85,B 0,C 180,E1 -15275.304,E2 -15275.304} C_VEL
LIN {X 0,Y 319.594,Z 509.302,A -85,B 0,C 180,E1 -15279.4,E2 -15279.4} C_VEL
LIN {X 0,Y 319.65,Z 509.292,A -85,B 0,C 180,E1 -15282.073,E2 -15282.073} C_VEL
LIN {X 0,Y 319.724,Z 509.282,A -85,B 0,C 180,E1 -15286.008,E2 -15286.008} C_VEL
LIN {X 0,Y 319.75,Z 509.274,A -85,B 0,C 180,E1 -15289.873,E2 -15289.873} C_VEL
LIN {X 0,Y 319.924,Z 509.253,A -85,B 0,C 180,E1 -15292.426,E2 -15292.426} C_VEL
LIN {X 0,Y 319.742,Z 509.279,A -85,B 0,C 180,E1 -15294.956,E2 -15294.956} C_VEL
LIN {X 0,Y 320.001,Z 509.251,A -85,B 0,C 180,E1 -15297.483,E2 -15297.483} C_VEL
LIN {X 0,Y 320.142,Z 509.224,A -85,B 0,C 180,E1 -15300,E2 -15300} C_VEL
LIN {X 0,Y 319.985,Z 509.244,A -85,B 0,C 180,E1 -15302.518,E2 -15302.518} C_VEL
LIN {X 0,Y 319.919,Z 509.256,A -85,B 0,C 180,E1 -15306.573,E2 -15306.573} C_VEL
LIN {X 0,Y 319.744,Z 509.275,A -85,B 0,C 180,E1 -15310.128,E2 -15310.128} C_VEL
LIN {X 0,Y 319.723,Z 509.278,A -85,B 0,C 180,E1 -15314.725,E2 -15314.725} C_VEL
LIN {X 0,Y 319.682,Z 509.287,A -85,B 0,C 180,E1 -15319.039,E2 -15319.039} C_VEL
LIN {X 0,Y 319.564,Z 509.299,A -85,B 0,C 180,E1 -15323.321,E2 -15323.321} C_VEL
LIN {X 0,Y 319.629,Z 509.291,A -85,B 0,C 180,E1 -15326.089,E2 -15326.089} C_VEL
LIN {X 0,Y 319.584,Z 509.298,A -85,B 0,C 180,E1 -15328.935,E2 -15328.935} C_VEL
LIN {X 0,Y 319.533,Z 509.306,A -85,B 0,C 180,E1 -15331.862,E2 -15331.862} C_VEL
LIN {X 0,Y 319.576,Z 509.296,A -85,B 0,C 180,E1 -15335.545,E2 -15335.545} C_VEL
LIN {X 0,Y 319.596,Z 509.297,A -85,B 0,C 180,E1 -15338.006,E2 -15338.006} C_VEL
LIN {X 0,Y 319.598,Z 509.302,A -85,B 0,C 180,E1 -15341.614,E2 -15341.614} C_VEL
LIN {X 0,Y 319.643,Z 509.291,A -85,B 0,C 180,E1 -15345.287,E2 -15345.287} C_VEL
LIN {X 0,Y 319.582,Z 509.297,A -85,B 0,C 180,E1 -15348.722,E2 -15348.722} C_VEL
LIN {X 0,Y 319.597,Z 509.297,A -85,B 0,C 180,E1 -15352.341,E2 -15352.341} C_VEL
LIN {X 0,Y 319.56,Z 509.3,A -85,B 0,C 180,E1 -15355.125,E2 -15355.125} C_VEL
LIN {X 0,Y 319.57,Z 509.302,A -85,B 0,C 180,E1 -15359.059,E2 -15359.059} C_VEL
LIN {X 0,Y 319.609,Z 509.293,A -85,B 0,C 180,E1 -15362.5,E2 -15362.5} C_VEL
LIN {X 0,Y 319.608,Z 509.296,A -85,B 0,C 180,E1 -15365.306,E2 -15365.306} C_VEL
LIN {X 0,Y 319.599,Z 509.298,A -85,B 0,C 180,E1 -15368.049,E2 -15368.049} C_VEL
LIN {X 0,Y 319.692,Z 509.283,A -85,B 0,C 180,E1 -15370.963,E2 -15370.963} C_VEL
LIN {X 0,Y 319.734,Z 509.281,A -85,B 0,C 180,E1 -15375.277,E2 -15375.277} C_VEL
LIN {X 0,Y 319.755,Z 509.278,A -85,B 0,C 180,E1 -15379.874,E2 -15379.874} C_VEL
LIN {X 0,Y 319.942,Z 509.257,A -85,B 0,C 180,E1 -15383.695,E2 -15383.695} C_VEL
LIN {X 0,Y 319.997,Z 509.251,A -85,B 0,C 180,E1 -15387.483,E2 -15387.483} C_VEL
LIN {X 0,Y 320.13,Z 509.232,A -85,B 0,C 180,E1 -15390.001,E2 -15390.001} C_VEL
LIN {X 0,Y 319.765,Z 509.277,A -85,B 0,C 180,E1 -15392.52,E2 -15392.52} C_VEL
LIN {X 0,Y 319.365,Z 509.33,A -85,B 0,C 180,E1 -15396.318,E2 -15396.318} C_VEL
LIN {X 0,Y 319.171,Z 509.947,A -85,B 0,C 180,E1 -15398.054,E2 -15398.054} C_VEL
LIN {X 0,Y 319.145,Z 510.015,A -85,B 0,C 180,E1 -15398.142,E2 -15398.142} C_VEL
LIN {X 0,Y 320.244,Z 513.231,A -85,B 0,C 180,E1 -15398.37,E2 -15398.37} C_VEL
LIN {X 0,Y 326.287,Z 528.523,A -85,B 0,C 180,E1 -15399.581,E2 -15399.581} C_VEL
LIN {X 0,Y 330.676,Z 541.808,A -85,B 0,C 180,E1 -15400.754,E2 -15400.754} C_VEL
LIN {X 0,Y 334.143,Z 554.075,A -85,B 0,C 180,E1 -15401.953,E2 -15401.953} C_VEL
LIN {X 0,Y 334.841,Z 557.116,A -85,B 0,C 180,E1 -15402.271,E2 -15402.271} C_VEL
LIN {X 0,Y 333.173,Z 570.708,A -85,B 0,C 180,E1 -15403.417,E2 -15403.417} C_VEL
LIN {X 0,Y 331.274,Z 583.591,A -85,B 0,C 180,E1 -15404.749,E2 -15404.749} C_VEL
LIN {X 0,Y 329.372,Z 595.352,A -85,B 0,C 180,E1 -15406.219,E2 -15406.219} C_VEL
LIN {X 0,Y 327.23,Z 607.103,A -85,B 0,C 180,E1 -15407.983,E2 -15407.983} C_VEL
LIN {X 0,Y 325.221,Z 617.693,A -85,B 0,C 180,E1 -15409.899,E2 -15409.899} C_VEL
LIN {X 0,Y 323.396,Z 627.394,A -85,B 0,C 180,E1 -15412.017,E2 -15412.017} C_VEL
LIN {X 0,Y 321.897,Z 635.042,A -85,B 0,C 180,E1 -15414.023,E2 -15414.023} C_VEL
LIN {X 0,Y 320.758,Z 641.56,A -85,B 0,C 180,E1 -15416.059,E2 -15416.059} C_VEL
LIN {X 0,Y 319.656,Z 647.805,A -85,B 0,C 180,E1 -15418.423,E2 -15418.423} C_VEL
LIN {X 0,Y 318.941,Z 652.699,A -85,B 0,C 180,E1 -15420.751,E2 -15420.751} C_VEL
LIN {X 0,Y 318.273,Z 657.018,A -85,B 0,C 180,E1 -15423.507,E2 -15423.507} C_VEL
LIN {X 0,Y 317.997,Z 658.867,A -85,B 0,C 180,E1 -15425.14,E2 -15425.14} C_VEL
LIN {X 0,Y 317.773,Z 660.539,A -85,B 0,C 180,E1 -15427.231,E2 -15427.231} C_VEL
LIN {X 0,Y 317.714,Z 661.55,A -85,B 0,C 180,E1 -15429.903,E2 -15429.903} C_VEL
LIN {X 0,Y 317.746,Z 661.56,A -85,B 0,C 180,E1 -15431.571,E2 -15431.571} C_VEL
LIN {X 0,Y 317.882,Z 661.085,A -85,B 0,C 180,E1 -15433.265,E2 -15433.265} C_VEL
LIN {X 0,Y 318.081,Z 660.026,A -85,B 0,C 180,E1 -15435.005,E2 -15435.005} C_VEL
LIN {X 0,Y 318.684,Z 657.303,A -85,B 0,C 180,E1 -15437.73,E2 -15437.73} C_VEL
LIN {X 0,Y 319.447,Z 653.372,A -85,B 0,C 180,E1 -15440.355,E2 -15440.355} C_VEL
LIN {X 0,Y 320.557,Z 648.023,A -85,B 0,C 180,E1 -15442.983,E2 -15442.983} C_VEL
LIN {X 0,Y 322.024,Z 641.627,A -85,B 0,C 180,E1 -15445.428,E2 -15445.428} C_VEL
LIN {X 0,Y 323.879,Z 633.855,A -85,B 0,C 180,E1 -15447.809,E2 -15447.809} C_VEL
LIN {X 0,Y 325.903,Z 625.11,A -85,B 0,C 180,E1 -15450,E2 -15450} C_VEL
LIN {X 0,Y 328.481,Z 614.034,A -85,B 0,C 180,E1 -15452.266,E2 -15452.266} C_VEL
LIN {X 0,Y 328.791,Z 612.549,A -85,B 0,C 180,E1 -15452.53,E2 -15452.53} C_VEL
LIN {X 0,Y 329.033,Z 608.587,A -85,B 0,C 180,E1 -15453.288,E2 -15453.288} C_VEL
LIN {X 0,Y 327.038,Z 596.681,A -85,B 0,C 180,E1 -15455.593,E2 -15455.593} C_VEL
LIN {X 0,Y 327.062,Z 592.266,A -85,B 0,C 180,E1 -15456.278,E2 -15456.278} C_VEL
LIN {X 0,Y 327.298,Z 590.707,A -85,B 0,C 180,E1 -15456.484,E2 -15456.484} C_VEL
LIN {X 0,Y 329.715,Z 578.084,A -85,B 0,C 180,E1 -15457.933,E2 -15457.933} C_VEL
LIN {X 0,Y 331.815,Z 565.464,A -85,B 0,C 180,E1 -15459.114,E2 -15459.114} C_VEL
LIN {X 0,Y 332.056,Z 562.465,A -85,B 0,C 180,E1 -15459.381,E2 -15459.381} C_VEL
LIN {X 0,Y 328.971,Z 550.893,A -85,B 0,C 180,E1 -15460.824,E2 -15460.824} C_VEL
LIN {X 0,Y 324.277,Z 537.976,A -85,B 0,C 180,E1 -15462.405,E2 -15462.405} C_VEL
LIN {X 0,Y 318.997,Z 526.462,A -85,B 0,C 180,E1 -15463.85,E2 -15463.85} C_VEL
LIN {X 0,Y 315.209,Z 519.36,A -85,B 0,C 180,E1 -15464.765,E2 -15464.765} C_VEL
LIN {X 0,Y 313.198,Z 515.883,A -85,B 0,C 180,E1 -15465.236,E2 -15465.236} C_VEL
LIN {X 0,Y 312.832,Z 514.445,A -85,B 0,C 180,E1 -15465.38,E2 -15465.38} C_VEL
LIN {X 0,Y 312.909,Z 512.991,A -85,B 0,C 180,E1 -15468.337,E2 -15468.337} C_VEL
LIN {X 0,Y 313.033,Z 511.245,A -85,B 0,C 180,E1 -15472.258,E2 -15472.258} C_VEL
LIN {X 0,Y 312.727,Z 510.272,A -85,B 0,C 180,E1 -15474.842,E2 -15474.842} C_VEL
LIN {X 0,Y 312.989,Z 510.123,A -85,B 0,C 180,E1 -15478.713,E2 -15478.713} C_VEL
LIN {X 0,Y 312.988,Z 510.122,A -85,B 0,C 180,E1 -15481.286,E2 -15481.286} C_VEL
LIN {X 0,Y 312.716,Z 510.155,A -85,B 0,C 180,E1 -15485.157,E2 -15485.157} C_VEL
LIN {X 0,Y 312.87,Z 510.137,A -85,B 0,C 180,E1 -15487.745,E2 -15487.745} C_VEL
LIN {X 0,Y 312.667,Z 510.16,A -85,B 0,C 180,E1 -15491.671,E2 -15491.671} C_VEL
LIN {X 0,Y 312.698,Z 510.157,A -85,B 0,C 180,E1 -15494.887,E2 -15494.887} C_VEL
LIN {X 0,Y 312.628,Z 510.165,A -85,B 0,C 180,E1 -15499.236,E2 -15499.236} C_VEL
LIN {X 0,Y 312.543,Z 510.177,A -85,B 0,C 180,E1 -15502.789,E2 -15502.789} C_VEL
LIN {X 0,Y 312.626,Z 510.352,A -85,B 0,C 180,E1 -15505.945,E2 -15505.945} C_VEL
LIN {X 0,Y 312.912,Z 512.35,A -85,B 0,C 180,E1 -15509.611,E2 -15509.611} C_VEL
LIN {X 0,Y 313.22,Z 514.295,A -85,B 0,C 180,E1 -15512.582,E2 -15512.582} C_VEL
LIN {X 0,Y 313.762,Z 517.109,A -85,B 0,C 180,E1 -15516.258,E2 -15516.258} C_VEL
LIN {X 0,Y 314.134,Z 519.344,A -85,B 0,C 180,E1 -15518.787,E2 -15518.787} C_VEL
LIN {X 0,Y 314.736,Z 523.088,A -85,B 0,C 180,E1 -15522.534,E2 -15522.534} C_VEL
LIN {X 0,Y 315.353,Z 527.32,A -85,B 0,C 180,E1 -15526.301,E2 -15526.301} C_VEL
LIN {X 0,Y 315.312,Z 529.5,A -85,B 0,C 180,E1 -15528.036,E2 -15528.036} C_VEL
LIN {X 0,Y 314.633,Z 534.091,A -85,B 0,C 180,E1 -15531.425,E2 -15531.425} C_VEL
LIN {X 0,Y 313.909,Z 538.937,A -85,B 0,C 180,E1 -15534.778,E2 -15534.778} C_VEL
LIN {X 0,Y 314.889,Z 542.341,A -85,B 0,C 180,E1 -15535.062,E2 -15535.062} C_VEL
LIN {X 0,Y 316.014,Z 544.908,A -85,B 0,C 180,E1 -15535.334,E2 -15535.334} C_VEL
LIN {X 0,Y 320.263,Z 556.954,A -85,B 0,C 180,E1 -15536.5,E2 -15536.5} C_VEL
LIN {X 0,Y 323.846,Z 569.97,A -85,B 0,C 180,E1 -15537.76,E2 -15537.76} C_VEL
LIN {X 0,Y 326.364,Z 582.939,A -85,B 0,C 180,E1 -15539.038,E2 -15539.038} C_VEL
LIN {X 0,Y 327.916,Z 596.786,A -85,B 0,C 180,E1 -15540.466,E2 -15540.466} C_VEL
LIN {X 0,Y 328.291,Z 605.888,A -85,B 0,C 180,E1 -15541.472,E2 -15541.472} C_VEL
LIN {X 0,Y 325.696,Z 619.398,A -85,B 0,C 180,E1 -15542.881,E2 -15542.881} C_VEL
LIN {X 0,Y 322.935,Z 632.409,A -85,B 0,C 180,E1 -15544.544,E2 -15544.544} C_VEL
LIN {X 0,Y 320.252,Z 644.301,A -85,B 0,C 180,E1 -15546.39,E2 -15546.39} C_VEL
LIN {X 0,Y 317.937,Z 654.678,A -85,B 0,C 180,E1 -15548.326,E2 -15548.326} C_VEL
LIN {X 0,Y 315.841,Z 664.387,A -85,B 0,C 180,E1 -15550.502,E2 -15550.502} C_VEL
LIN {X 0,Y 314.078,Z 672.756,A -85,B 0,C 180,E1 -15552.753,E2 -15552.753} C_VEL
LIN {X 0,Y 312.554,Z 680.261,A -85,B 0,C 180,E1 -15555.213,E2 -15555.213} C_VEL
LIN {X 0,Y 311.698,Z 686.215,A -85,B 0,C 180,E1 -15557.631,E2 -15557.631} C_VEL
LIN {X 0,Y 311.083,Z 691.317,A -85,B 0,C 180,E1 -15560.244,E2 -15560.244} C_VEL
LIN {X 0,Y 310.887,Z 694.328,A -85,B 0,C 180,E1 -15562.204,E2 -15562.204} C_VEL
LIN {X 0,Y 310.801,Z 697.17,A -85,B 0,C 180,E1 -15564.81,E2 -15564.81} C_VEL
LIN {X 0,Y 310.83,Z 698.811,A -85,B 0,C 180,E1 -15567.408,E2 -15567.408} C_VEL
LIN {X 0,Y 311.065,Z 699.288,A -85,B 0,C 180,E1 -15569.999,E2 -15569.999} C_VEL
LIN {X 0,Y 310.834,Z 698.555,A -85,B 0,C 180,E1 -15572.591,E2 -15572.591} C_VEL
LIN {X 0,Y 310.851,Z 696.624,A -85,B 0,C 180,E1 -15575.188,E2 -15575.188} C_VEL
LIN {X 0,Y 310.93,Z 693.405,A -85,B 0,C 180,E1 -15577.794,E2 -15577.794} C_VEL
LIN {X 0,Y 311.165,Z 688.868,A -85,B 0,C 180,E1 -15580.409,E2 -15580.409} C_VEL
LIN {X 0,Y 311.837,Z 682.918,A -85,B 0,C 180,E1 -15583.024,E2 -15583.024} C_VEL
LIN {X 0,Y 312.686,Z 677.206,A -85,B 0,C 180,E1 -15585.059,E2 -15585.059} C_VEL
LIN {X 0,Y 314.123,Z 668.589,A -85,B 0,C 180,E1 -15587.579,E2 -15587.579} C_VEL
LIN {X 0,Y 315.977,Z 659.178,A -85,B 0,C 180,E1 -15589.827,E2 -15589.827} C_VEL
LIN {X 0,Y 317.88,Z 648.809,A -85,B 0,C 180,E1 -15591.883,E2 -15591.883} C_VEL
LIN {X 0,Y 319.867,Z 638.237,A -85,B 0,C 180,E1 -15593.638,E2 -15593.638} C_VEL
LIN {X 0,Y 322.121,Z 625.796,A -85,B 0,C 180,E1 -15595.351,E2 -15595.351} C_VEL
LIN {X 0,Y 324.622,Z 612.138,A -85,B 0,C 180,E1 -15596.867,E2 -15596.867} C_VEL
LIN {X 0,Y 325.784,Z 604.578,A -85,B 0,C 180,E1 -15597.582,E2 -15597.582} C_VEL
LIN {X 0,Y 324.376,Z 591.376,A -85,B 0,C 180,E1 -15598.902,E2 -15598.902} C_VEL
LIN {X 0,Y 321.875,Z 576.302,A -85,B 0,C 180,E1 -15600.223,E2 -15600.223} C_VEL
LIN {X 0,Y 318.4,Z 560.952,A -85,B 0,C 180,E1 -15601.393,E2 -15601.393} C_VEL
LIN {X 0,Y 314.087,Z 545.783,A -85,B 0,C 180,E1 -15602.39,E2 -15602.39} C_VEL
LIN {X 0,Y 313.37,Z 542.751,A -85,B 0,C 180,E1 -15602.563,E2 -15602.563} C_VEL
LIN {X 0,Y 314.114,Z 536.842,A -85,B 0,C 180,E1 -15606.345,E2 -15606.345} C_VEL
LIN {X 0,Y 315.004,Z 530.85,A -85,B 0,C 180,E1 -15610.315,E2 -15610.315} C_VEL
LIN {X 0,Y 315.37,Z 527.432,A -85,B 0,C 180,E1 -15612.659,E2 -15612.659} C_VEL
LIN {X 0,Y 314.94,Z 523.503,A -85,B 0,C 180,E1 -15615.567,E2 -15615.567} C_VEL
LIN {X 0,Y 313.937,Z 518.459,A -85,B 0,C 180,E1 -15619.563,E2 -15619.563} C_VEL
LIN {X 0,Y 313.288,Z 514.718,A -85,B 0,C 180,E1 -15622.722,E2 -15622.722} C_VEL
LIN {X 0,Y 312.522,Z 510.179,A -85,B 0,C 180,E1 -15626.866,E2 -15626.866} C_VEL
LIN {X 0,Y 312.541,Z 510.175,A -85,B 0,C 180,E1 -15630.35,E2 -15630.35} C_VEL
LIN {X 0,Y 312.594,Z 510.171,A -85,B 0,C 180,E1 -15634.064,E2 -15634.064} C_VEL
LIN {X 0,Y 312.555,Z 510.18,A -85,B 0,C 180,E1 -15637.527,E2 -15637.527} C_VEL
LIN {X 0,Y 312.629,Z 510.169,A -85,B 0,C 180,E1 -15641.656,E2 -15641.656} C_VEL
LIN {X 0,Y 312.685,Z 510.162,A -85,B 0,C 180,E1 -15645.686,E2 -15645.686} C_VEL
LIN {X 0,Y 312.695,Z 510.154,A -85,B 0,C 180,E1 -15649.642,E2 -15649.642} C_VEL
LIN {X 0,Y 312.863,Z 510.132,A -85,B 0,C 180,E1 -15652.255,E2 -15652.255} C_VEL
LIN {X 0,Y 312.712,Z 510.154,A -85,B 0,C 180,E1 -15654.843,E2 -15654.843} C_VEL
LIN {X 0,Y 312.945,Z 510.13,A -85,B 0,C 180,E1 -15657.426,E2 -15657.426} C_VEL
LIN {X 0,Y 313.095,Z 510.1,A -85,B 0,C 180,E1 -15660.001,E2 -15660.001} C_VEL
LIN {X 0,Y 312.932,Z 510.122,A -85,B 0,C 180,E1 -15662.575,E2 -15662.575} C_VEL
LIN {X 0,Y 312.886,Z 510.132,A -85,B 0,C 180,E1 -15666.552,E2 -15666.552} C_VEL
LIN {X 0,Y 312.759,Z 510.149,A -85,B 0,C 180,E1 -15669.051,E2 -15669.051} C_VEL
LIN {X 0,Y 312.625,Z 510.157,A -85,B 0,C 180,E1 -15672.992,E2 -15672.992} C_VEL
LIN {X 0,Y 312.631,Z 510.168,A -85,B 0,C 180,E1 -15675.651,E2 -15675.651} C_VEL
LIN {X 0,Y 312.623,Z 510.168,A -85,B 0,C 180,E1 -15679.237,E2 -15679.237} C_VEL
LIN {X 0,Y 312.539,Z 510.17,A -85,B 0,C 180,E1 -15682.79,E2 -15682.79} C_VEL
LIN {X 0,Y 312.597,Z 510.167,A -85,B 0,C 180,E1 -15685.937,E2 -15685.937} C_VEL
LIN {X 0,Y 312.541,Z 510.18,A -85,B 0,C 180,E1 -15689.651,E2 -15689.651} C_VEL
LIN {X 0,Y 312.515,Z 510.177,A -85,B 0,C 180,E1 -15693.69,E2 -15693.69} C_VEL
LIN {X 0,Y 312.549,Z 510.172,A -85,B 0,C 180,E1 -15697.383,E2 -15697.383} C_VEL
LIN {X 0,Y 312.532,Z 510.177,A -85,B 0,C 180,E1 -15700.703,E2 -15700.703} C_VEL
LIN {X 0,Y 312.592,Z 510.166,A -85,B 0,C 180,E1 -15704.185,E2 -15704.185} C_VEL
LIN {X 0,Y 312.555,Z 510.175,A -85,B 0,C 180,E1 -15707.905,E2 -15707.905} C_VEL
LIN {X 0,Y 312.557,Z 510.177,A -85,B 0,C 180,E1 -15711.906,E2 -15711.906} C_VEL
LIN {X 0,Y 312.506,Z 510.18,A -85,B 0,C 180,E1 -15715.791,E2 -15715.791} C_VEL
LIN {X 0,Y 312.523,Z 510.179,A -85,B 0,C 180,E1 -15718.855,E2 -15718.855} C_VEL
LIN {X 0,Y 312.575,Z 510.173,A -85,B 0,C 180,E1 -15721.826,E2 -15721.826} C_VEL
LIN {X 0,Y 312.588,Z 510.168,A -85,B 0,C 180,E1 -15724.712,E2 -15724.712} C_VEL
LIN {X 0,Y 312.59,Z 510.175,A -85,B 0,C 180,E1 -15727.53,E2 -15727.53} C_VEL
LIN {X 0,Y 312.641,Z 510.167,A -85,B 0,C 180,E1 -15731.658,E2 -15731.658} C_VEL
LIN {X 0,Y 312.697,Z 510.158,A -85,B 0,C 180,E1 -15735.687,E2 -15735.687} C_VEL
LIN {X 0,Y 312.701,Z 510.158,A -85,B 0,C 180,E1 -15739.643,E2 -15739.643} C_VEL
LIN {X 0,Y 312.898,Z 510.135,A -85,B 0,C 180,E1 -15743.553,E2 -15743.553} C_VEL
LIN {X 0,Y 312.943,Z 510.129,A -85,B 0,C 180,E1 -15747.426,E2 -15747.426} C_VEL
LIN {X 0,Y 313.082,Z 510.11,A -85,B 0,C 180,E1 -15750.001,E2 -15750.001} C_VEL
LIN {X 0,Y 312.693,Z 510.158,A -85,B 0,C 180,E1 -15752.577,E2 -15752.577} C_VEL
LIN {X 0,Y 312.298,Z 510.21,A -85,B 0,C 180,E1 -15756.461,E2 -15756.461} C_VEL
LIN {X 0,Y 312.198,Z 510.502,A -85,B 0,C 180,E1 -15757.462,E2 -15757.462} C_VEL
LIN {X 0,Y 313.213,Z 513.478,A -85,B 0,C 180,E1 -15757.669,E2 -15757.669} C_VEL
LIN {X 0,Y 319.367,Z 529.059,A -85,B 0,C 180,E1 -15758.949,E2 -15758.949} C_VEL
LIN {X 0,Y 323.861,Z 542.219,A -85,B 0,C 180,E1 -15760.154,E2 -15760.154} C_VEL
LIN {X 0,Y 327.604,Z 555.817,A -85,B 0,C 180,E1 -15761.53,E2 -15761.53} C_VEL
LIN {X 0,Y 328.33,Z 558.838,A -85,B 0,C 180,E1 -15761.861,E2 -15761.861} C_VEL
LIN {X 0,Y 326.489,Z 572.581,A -85,B 0,C 180,E1 -15763.063,E2 -15763.063} C_VEL
LIN {X 0,Y 324.513,Z 585.226,A -85,B 0,C 180,E1 -15764.422,E2 -15764.422} C_VEL
LIN {X 0,Y 322.514,Z 597.052,A -85,B 0,C 180,E1 -15765.961,E2 -15765.961} C_VEL
LIN {X 0,Y 320.383,Z 608.356,A -85,B 0,C 180,E1 -15767.72,E2 -15767.72} C_VEL
LIN {X 0,Y 318.315,Z 618.827,A -85,B 0,C 180,E1 -15769.676,E2 -15769.676} C_VEL
LIN {X 0,Y 316.552,Z 627.856,A -85,B 0,C 180,E1 -15771.698,E2 -15771.698} C_VEL
LIN {X 0,Y 314.779,Z 636.588,A -85,B 0,C 180,E1 -15774.057,E2 -15774.057} C_VEL
LIN {X 0,Y 313.342,Z 644.345,A -85,B 0,C 180,E1 -15776.653,E2 -15776.653} C_VEL
LIN {X 0,Y 312.303,Z 650.253,A -85,B 0,C 180,E1 -15779.14,E2 -15779.14} C_VEL
LIN {X 0,Y 311.552,Z 655.463,A -85,B 0,C 180,E1 -15782.013,E2 -15782.013} C_VEL
LIN {X 0,Y 311,Z 658.566,A -85,B 0,C 180,E1 -15784.399,E2 -15784.399} C_VEL
LIN {X 0,Y 310.785,Z 660.12,A -85,B 0,C 180,E1 -15786.012,E2 -15786.012} C_VEL
LIN {X 0,Y 310.669,Z 661.237,A -85,B 0,C 180,E1 -15787.647,E2 -15787.647} C_VEL
LIN {X 0,Y 310.621,Z 661.941,A -85,B 0,C 180,E1 -15789.71,E2 -15789.71} C_VEL
LIN {X 0,Y 310.665,Z 661.993,A -85,B 0,C 180,E1 -15791.707,E2 -15791.707} C_VEL
LIN {X 0,Y 310.938,Z 660.928,A -85,B 0,C 180,E1 -15794.481,E2 -15794.481} C_VEL
LIN {X 0,Y 311.222,Z 659.584,A -85,B 0,C 180,E1 -15796.271,E2 -15796.271} C_VEL
LIN {X 0,Y 312.032,Z 656.088,A -85,B 0,C 180,E1 -15799.218,E2 -15799.218} C_VEL
LIN {X 0,Y 312.939,Z 651.691,A -85,B 0,C 180,E1 -15801.816,E2 -15801.816} C_VEL
LIN {X 0,Y 314.344,Z 645.793,A -85,B 0,C 180,E1 -15804.457,E2 -15804.457} C_VEL
LIN {X 0,Y 316.017,Z 638.88,A -85,B 0,C 180,E1 -15806.9,E2 -15806.9} C_VEL
LIN {X 0,Y 317.894,Z 631.347,A -85,B 0,C 180,E1 -15809.069,E2 -15809.069} C_VEL
LIN {X 0,Y 320.321,Z 621.691,A -85,B 0,C 180,E1 -15811.356,E2 -15811.356} C_VEL
LIN {X 0,Y 322.8,Z 611.232,A -85,B 0,C 180,E1 -15813.401,E2 -15813.401} C_VEL
LIN {X 0,Y 325.281,Z 600.377,A -85,B 0,C 180,E1 -15815.154,E2 -15815.154} C_VEL
LIN {X 0,Y 327.298,Z 590.707,A -85,B 0,C 180,E1 -15816.484,E2 -15816.484} C_VEL
LIN {X 0,Y 327.665,Z 586.049,A -85,B 0,C 180,E1 -15817.115,E2 -15817.115} C_VEL
LIN {X 0,Y 325.826,Z 572.334,A -85,B 0,C 180,E1 -15819.093,E2 -15819.093} C_VEL
LIN {X 0,Y 325.829,Z 566.538,A -85,B 0,C 180,E1 -15819.739,E2 -15819.739} C_VEL
LIN {X 0,Y 325.963,Z 565.676,A -85,B 0,C 180,E1 -15819.818,E2 -15819.818} C_VEL
LIN {X 0,Y 324.96,Z 560.238,A -85,B 0,C 180,E1 -15820.495,E2 -15820.495} C_VEL
LIN {X 0,Y 321.575,Z 548.921,A -85,B 0,C 180,E1 -15821.966,E2 -15821.966} C_VEL
LIN {X 0,Y 317.144,Z 537.344,A -85,B 0,C 180,E1 -15823.489,E2 -15823.489} C_VEL
LIN {X 0,Y 311.994,Z 526.773,A -85,B 0,C 180,E1 -15824.923,E2 -15824.923} C_VEL
LIN {X 0,Y 307.954,Z 519.316,A -85,B 0,C 180,E1 -15825.966,E2 -15825.966} C_VEL
LIN {X 0,Y 306.217,Z 516.481,A -85,B 0,C 180,E1 -15826.393,E2 -15826.393} C_VEL
LIN {X 0,Y 305.862,Z 515.065,A -85,B 0,C 180,E1 -15826.546,E2 -15826.546} C_VEL
LIN {X 0,Y 306.04,Z 513.08,A -85,B 0,C 180,E1 -15830.916,E2 -15830.916} C_VEL
LIN {X 0,Y 306.002,Z 512.09,A -85,B 0,C 180,E1 -15833.405,E2 -15833.405} C_VEL
LIN {X 0,Y 305.885,Z 511.009,A -85,B 0,C 180,E1 -15837.366,E2 -15837.366} C_VEL
LIN {X 0,Y 306.053,Z 510.986,A -85,B 0,C 180,E1 -15839.999,E2 -15839.999} C_VEL
LIN {X 0,Y 305.884,Z 511.009,A -85,B 0,C 180,E1 -15842.633,E2 -15842.633} C_VEL
LIN {X 0,Y 305.85,Z 511.012,A -85,B 0,C 180,E1 -15846.597,E2 -15846.597} C_VEL
LIN {X 0,Y 305.734,Z 511.024,A -85,B 0,C 180,E1 -15849.259,E2 -15849.259} C_VEL
LIN {X 0,Y 305.586,Z 511.041,A -85,B 0,C 180,E1 -15853.296,E2 -15853.296} C_VEL
LIN {X 0,Y 305.591,Z 511.043,A -85,B 0,C 180,E1 -15856.02,E2 -15856.02} C_VEL
LIN {X 0,Y 305.574,Z 511.044,A -85,B 0,C 180,E1 -15859.444,E2 -15859.444} C_VEL
LIN {X 0,Y 305.488,Z 511.055,A -85,B 0,C 180,E1 -15863.041,E2 -15863.041} C_VEL
LIN {X 0,Y 305.72,Z 511.941,A -85,B 0,C 180,E1 -15865.898,E2 -15865.898} C_VEL
LIN {X 0,Y 305.958,Z 513.684,A -85,B 0,C 180,E1 -15869.206,E2 -15869.206} C_VEL
LIN {X 0,Y 306.398,Z 516.426,A -85,B 0,C 180,E1 -15873.401,E2 -15873.401} C_VEL
LIN {X 0,Y 306.865,Z 518.999,A -85,B 0,C 180,E1 -15876.718,E2 -15876.718} C_VEL
LIN {X 0,Y 307.331,Z 521.77,A -85,B 0,C 180,E1 -15879.814,E2 -15879.814} C_VEL
LIN {X 0,Y 307.862,Z 525.19,A -85,B 0,C 180,E1 -15883.223,E2 -15883.223} C_VEL
LIN {X 0,Y 308.341,Z 528.127,A -85,B 0,C 180,E1 -15885.886,E2 -15885.886} C_VEL
LIN {X 0,Y 308.198,Z 531.45,A -85,B 0,C 180,E1 -15888.601,E2 -15888.601} C_VEL
LIN {X 0,Y 307.521,Z 535.861,A -85,B 0,C 180,E1 -15891.899,E2 -15891.899} C_VEL
LIN {X 0,Y 307.113,Z 538.469,A -85,B 0,C 180,E1 -15893.673,E2 -15893.673} C_VEL
LIN {X 0,Y 308.104,Z 541.746,A -85,B 0,C 180,E1 -15893.964,E2 -15893.964} C_VEL
LIN {X 0,Y 309.245,Z 544.314,A -85,B 0,C 180,E1 -15894.262,E2 -15894.262} C_VEL
LIN {X 0,Y 313.754,Z 556.559,A -85,B 0,C 180,E1 -15895.544,E2 -15895.544} C_VEL
LIN {X 0,Y 317.479,Z 570.11,A -85,B 0,C 180,E1 -15896.938,E2 -15896.938} C_VEL
LIN {X 0,Y 320.135,Z 583.648,A -85,B 0,C 180,E1 -15898.347,E2 -15898.347} C_VEL
LIN {X 0,Y 321.595,Z 597.325,A -85,B 0,C 180,E1 -15899.826,E2 -15899.826} C_VEL
LIN {X 0,Y 321.94,Z 606.699,A -85,B 0,C 180,E1 -15900.909,E2 -15900.909} C_VEL
LIN {X 0,Y 319.094,Z 620.876,A -85,B 0,C 180,E1 -15902.45,E2 -15902.45} C_VEL
LIN {X 0,Y 316.277,Z 633.564,A -85,B 0,C 180,E1 -15904.145,E2 -15904.145} C_VEL
LIN {X 0,Y 313.732,Z 644.296,A -85,B 0,C 180,E1 -15905.869,E2 -15905.869} C_VEL
LIN {X 0,Y 311.137,Z 655.204,A -85,B 0,C 180,E1 -15907.976,E2 -15907.976} C_VEL
LIN {X 0,Y 309.113,Z 664.196,A -85,B 0,C 180,E1 -15910.059,E2 -15910.059} C_VEL
LIN {X 0,Y 307.201,Z 672.527,A -85,B 0,C 180,E1 -15912.354,E2 -15912.354} C_VEL
LIN {X 0,Y 305.531,Z 680.447,A -85,B 0,C 180,E1 -15915.039,E2 -15915.039} C_VEL
LIN {X 0,Y 304.501,Z 687.312,A -85,B 0,C 180,E1 -15918.011,E2 -15918.011} C_VEL
LIN {X 0,Y 303.933,Z 692.064,A -85,B 0,C 180,E1 -15920.684,E2 -15920.684} C_VEL
LIN {X 0,Y 303.722,Z 695.531,A -85,B 0,C 180,E1 -15923.356,E2 -15923.356} C_VEL
LIN {X 0,Y 303.742,Z 697.743,A -85,B 0,C 180,E1 -15926.019,E2 -15926.019} C_VEL
LIN {X 0,Y 303.858,Z 698.772,A -85,B 0,C 180,E1 -15928.674,E2 -15928.674} C_VEL
LIN {X 0,Y 303.976,Z 698.849,A -85,B 0,C 180,E1 -15929.999,E2 -15929.999} C_VEL
LIN {X 0,Y 303.751,Z 698.086,A -85,B 0,C 180,E1 -15932.652,E2 -15932.652} C_VEL
LIN {X 0,Y 303.771,Z 696.132,A -85,B 0,C 180,E1 -15935.309,E2 -15935.309} C_VEL
LIN {X 0,Y 303.84,Z 692.885,A -85,B 0,C 180,E1 -15937.977,E2 -15937.977} C_VEL
LIN {X 0,Y 304.109,Z 688.312,A -85,B 0,C 180,E1 -15940.653,E2 -15940.653} C_VEL
LIN {X 0,Y 304.835,Z 682.322,A -85,B 0,C 180,E1 -15943.329,E2 -15943.329} C_VEL
LIN {X 0,Y 306.056,Z 674.762,A -85,B 0,C 180,E1 -15945.994,E2 -15945.994} C_VEL
LIN {X 0,Y 307.459,Z 666.647,A -85,B 0,C 180,E1 -15948.318,E2 -15948.318} C_VEL
LIN {X 0,Y 309.464,Z 656.924,A -85,B 0,C 180,E1 -15950.609,E2 -15950.609} C_VEL
LIN {X 0,Y 311.373,Z 646.983,A -85,B 0,C 180,E1 -15952.562,E2 -15952.562} C_VEL
LIN {X 0,Y 313.696,Z 635.205,A -85,B 0,C 180,E1 -15954.485,E2 -15954.485} C_VEL
LIN {X 0,Y 316.123,Z 622.24,A -85,B 0,C 180,E1 -15956.221,E2 -15956.221} C_VEL
LIN {X 0,Y 318.659,Z 608.286,A -85,B 0,C 180,E1 -15957.724,E2 -15957.724} C_VEL
LIN {X 0,Y 319.099,Z 605.303,A -85,B 0,C 180,E1 -15958.016,E2 -15958.016} C_VEL
LIN {X 0,Y 317.762,Z 592.567,A -85,B 0,C 180,E1 -15959.338,E2 -15959.338} C_VEL
LIN {X 0,Y 315.378,Z 577.866,A -85,B 0,C 180,E1 -15960.684,E2 -15960.684} C_VEL
LIN {X 0,Y 312.205,Z 563.416,A -85,B 0,C 180,E1 -15961.844,E2 -15961.844} C_VEL
LIN {X 0,Y 308.149,Z 548.68,A -85,B 0,C 180,E1 -15962.885,E2 -15962.885} C_VEL
LIN {X 0,Y 306.433,Z 542.342,A -85,B 0,C 180,E1 -15963.303,E2 -15963.303} C_VEL
LIN {X 0,Y 307.152,Z 537.017,A -85,B 0,C 180,E1 -15966.79,E2 -15966.79} C_VEL
LIN {X 0,Y 308,Z 531.609,A -85,B 0,C 180,E1 -15970.449,E2 -15970.449} C_VEL
LIN {X 0,Y 308.326,Z 527.814,A -85,B 0,C 180,E1 -15973.164,E2 -15973.164} C_VEL
LIN {X 0,Y 307.855,Z 524.227,A -85,B 0,C 180,E1 -15975.886,E2 -15975.886} C_VEL
LIN {X 0,Y 307.076,Z 520.307,A -85,B 0,C 180,E1 -15979.046,E2 -15979.046} C_VEL
LIN {X 0,Y 306.533,Z 517.121,A -85,B 0,C 180,E1 -15981.755,E2 -15981.755} C_VEL
LIN {X 0,Y 305.762,Z 512.607,A -85,B 0,C 180,E1 -15985.837,E2 -15985.837} C_VEL
LIN {X 0,Y 305.466,Z 511.058,A -85,B 0,C 180,E1 -15987.467,E2 -15987.467} C_VEL
LIN {X 0,Y 305.52,Z 511.053,A -85,B 0,C 180,E1 -15991.114,E2 -15991.114} C_VEL
LIN {X 0,Y 305.563,Z 511.047,A -85,B 0,C 180,E1 -15994.088,E2 -15994.088} C_VEL
LIN {X 0,Y 305.473,Z 511.057,A -85,B 0,C 180,E1 -15998.401,E2 -15998.401} C_VEL
LIN {X 0,Y 305.581,Z 511.047,A -85,B 0,C 180,E1 -16001.218,E2 -16001.218} C_VEL
LIN {X 0,Y 305.64,Z 511.039,A -85,B 0,C 180,E1 -16005.349,E2 -16005.349} C_VEL
LIN {X 0,Y 305.632,Z 511.036,A -85,B 0,C 180,E1 -16009.4,E2 -16009.4} C_VEL
LIN {X 0,Y 305.804,Z 511.012,A -85,B 0,C 180,E1 -16012.075,E2 -16012.075} C_VEL
LIN {X 0,Y 305.683,Z 511.03,A -85,B 0,C 180,E1 -16014.724,E2 -16014.724} C_VEL
LIN {X 0,Y 305.952,Z 510.993,A -85,B 0,C 180,E1 -16018.684,E2 -16018.684} C_VEL
LIN {X 0,Y 305.951,Z 510.99,A -85,B 0,C 180,E1 -16021.317,E2 -16021.317} C_VEL
LIN {X 0,Y 305.684,Z 511.032,A -85,B 0,C 180,E1 -16025.277,E2 -16025.277} C_VEL
LIN {X 0,Y 305.79,Z 511.017,A -85,B 0,C 180,E1 -16027.927,E2 -16027.927} C_VEL
LIN {X 0,Y 305.595,Z 511.032,A -85,B 0,C 180,E1 -16031.946,E2 -16031.946} C_VEL
LIN {X 0,Y 305.63,Z 511.033,A -85,B 0,C 180,E1 -16035.036,E2 -16035.036} C_VEL
LIN {X 0,Y 305.569,Z 511.048,A -85,B 0,C 180,E1 -16039.446,E2 -16039.446} C_VEL
LIN {X 0,Y 305.484,Z 511.049,A -85,B 0,C 180,E1 -16043.042,E2 -16043.042} C_VEL
LIN {X 0,Y 305.542,Z 511.044,A -85,B 0,C 180,E1 -16046.228,E2 -16046.228} C_VEL
LIN {X 0,Y 305.491,Z 511.055,A -85,B 0,C 180,E1 -16049.051,E2 -16049.051} C_VEL
LIN {X 0,Y 305.443,Z 511.059,A -85,B 0,C 180,E1 -16051.953,E2 -16051.953} C_VEL
LIN {X 0,Y 305.459,Z 511.052,A -85,B 0,C 180,E1 -16055.114,E2 -16055.114} C_VEL
LIN {X 0,Y 305.49,Z 511.052,A -85,B 0,C 180,E1 -16058.541,E2 -16058.541} C_VEL
LIN {X 0,Y 305.519,Z 511.05,A -85,B 0,C 180,E1 -16062.601,E2 -16062.601} C_VEL
LIN {X 0,Y 305.532,Z 511.041,A -85,B 0,C 180,E1 -16066.366,E2 -16066.366} C_VEL
LIN {X 0,Y 305.499,Z 511.057,A -85,B 0,C 180,E1 -16069.901,E2 -16069.901} C_VEL
LIN {X 0,Y 305.501,Z 511.054,A -85,B 0,C 180,E1 -16073.628,E2 -16073.628} C_VEL
LIN {X 0,Y 305.464,Z 511.054,A -85,B 0,C 180,E1 -16076.485,E2 -16076.485} C_VEL
LIN {X 0,Y 305.496,Z 511.055,A -85,B 0,C 180,E1 -16080.951,E2 -16080.951} C_VEL
LIN {X 0,Y 305.573,Z 511.043,A -85,B 0,C 180,E1 -16084.089,E2 -16084.089} C_VEL
LIN {X 0,Y 305.503,Z 511.052,A -85,B 0,C 180,E1 -16088.404,E2 -16088.404} C_VEL
LIN {X 0,Y 305.593,Z 511.04,A -85,B 0,C 180,E1 -16091.219,E2 -16091.219} C_VEL
LIN {X 0,Y 305.652,Z 511.035,A -85,B 0,C 180,E1 -16095.35,E2 -16095.35} C_VEL
LIN {X 0,Y 305.639,Z 511.04,A -85,B 0,C 180,E1 -16099.401,E2 -16099.401} C_VEL
LIN {X 0,Y 305.776,Z 511.021,A -85,B 0,C 180,E1 -16102.074,E2 -16102.074} C_VEL
LIN {X 0,Y 305.69,Z 511.027,A -85,B 0,C 180,E1 -16104.724,E2 -16104.724} C_VEL
LIN {X 0,Y 305.963,Z 510.996,A -85,B 0,C 180,E1 -16108.684,E2 -16108.684} C_VEL
LIN {X 0,Y 305.904,Z 511.004,A -85,B 0,C 180,E1 -16111.317,E2 -16111.317} C_VEL
LIN {X 0,Y 305.376,Z 511.072,A -85,B 0,C 180,E1 -16115.283,E2 -16115.283} C_VEL
LIN {X 0,Y 305.21,Z 511.104,A -85,B 0,C 180,E1 -16116.736,E2 -16116.736} C_VEL
LIN {X 0,Y 306.305,Z 514.139,A -85,B 0,C 180,E1 -16116.96,E2 -16116.96} C_VEL
LIN {X 0,Y 312.11,Z 528.578,A -85,B 0,C 180,E1 -16118.199,E2 -16118.199} C_VEL
LIN {X 0,Y 316.718,Z 541.88,A -85,B 0,C 180,E1 -16119.454,E2 -16119.454} C_VEL
LIN {X 0,Y 320.64,Z 555.781,A -85,B 0,C 180,E1 -16120.893,E2 -16120.893} C_VEL
LIN {X 0,Y 321.626,Z 559.746,A -85,B 0,C 180,E1 -16121.342,E2 -16121.342} C_VEL
LIN {X 0,Y 321.476,Z 563.374,A -85,B 0,C 180,E1 -16121.667,E2 -16121.667} C_VEL
LIN {X 0,Y 319.616,Z 575.955,A -85,B 0,C 180,E1 -16122.846,E2 -16122.846} C_VEL
LIN {X 0,Y 317.279,Z 589.702,A -85,B 0,C 180,E1 -16124.43,E2 -16124.43} C_VEL
LIN {X 0,Y 315.059,Z 602.146,A -85,B 0,C 180,E1 -16126.202,E2 -16126.202} C_VEL
LIN {X 0,Y 312.898,Z 612.66,A -85,B 0,C 180,E1 -16127.99,E2 -16127.99} C_VEL
LIN {X 0,Y 310.703,Z 623.345,A -85,B 0,C 180,E1 -16130.179,E2 -16130.179} C_VEL
LIN {X 0,Y 308.838,Z 632.341,A -85,B 0,C 180,E1 -16132.419,E2 -16132.419} C_VEL
LIN {X 0,Y 307.093,Z 640.987,A -85,B 0,C 180,E1 -16135.049,E2 -16135.049} C_VEL
LIN {X 0,Y 305.964,Z 647.065,A -85,B 0,C 180,E1 -16137.349,E2 -16137.349} C_VEL
LIN {X 0,Y 305.087,Z 652.087,A -85,B 0,C 180,E1 -16139.687,E2 -16139.687} C_VEL
